TYPE UDT 31
VERSION : 0.0
  STRUCT
   A_FD_OR : BYTE ;	//Feedrate override
   A_DriveEnable : BOOL ;	//Drive test movement enable
   A_AckFixedStop : BOOL ;	//Acknowledge fixed stop reached
   A_SensorFixedStop : BOOL ;	//Sensor fixed stop
   A_ASpDisable : BOOL ;	//Axis/spindle disable
   A_Follow_upMode : BOOL ;	//Follow-up mode
   A_PosMeas1 : BOOL ;	//Position measuring system 1
   A_PosMeas2 : BOOL ;	//Position measuring system 2
   A_ORactive : BOOL ;	//Override active
   A_SWCam : BOOL ;	//SW cam activation
   A_ContrEnable : BOOL ;	//Controller enable
   A_DelDTGSpReset : BOOL ;	//Delete distance to go/Spindle-Reset
   A_Clamp : BOOL ;	//Clamping in progress
   A_RefVal1 : BOOL ;	//Reference point value 1
   A_RefVal2 : BOOL ;	//Reference point value 2
   A_RefVal3 : BOOL ;	//Reference point value 3
   A_RefVal4 : BOOL ;	//Reference point value 4
   A_ExtZO : BOOL ;	//Import external ZO
   A_EnabTravFixedStop : BOOL ;	//Enable travel to fixed stop
   A_FixedFD1 : BOOL ;	//Activate fixed feed 1
   A_FixedFD2 : BOOL ;	//Activate fixed feed 2
   A_FixedFD3 : BOOL ;	//Activate fixed feed 3
   A_FixedFD4 : BOOL ;	//Activate fixed feed 4
   A_VelocSpeedLimit : BOOL ;	//Velocity/spindle speed limitation
   A_PrgtestAxRel : BOOL ;	// Program test axis/spindle release
   A_HW1 : BOOL ;	//Activate handwheel 1
   A_HW2 : BOOL ;	//Activate handwheel 2
   A_HW3 : BOOL ;	//Activate handwheel 3
   A_FDSpStop : BOOL ;	//Feed stop/spindle stop
   A_Disable : BOOL ;	//Traversing key disable
   A_RapidTrOR : BOOL ;	//Rapid traverse override
   A_Minus : BOOL ;	//Traversing key minus
   A_Plus : BOOL ;	//Traversing key plus
   A_INC1 : BOOL ;	//INC1
   A_INC10 : BOOL ;	//INC10
   A_INC100 : BOOL ;	//INC100
   A_INC1000 : BOOL ;	//INC1000
   A_INC10000 : BOOL ;	//INC10000
   A_INCVar : BOOL ;	//INC variable
   A_OEMAxis : BYTE ;	//OEM axis signals
   A_InvHWDirOfRot : BOOL ;	// Inverting handwheel direction of rotation
   f7_1 : BOOL ;
   f7_2 : BOOL ;
   f7_3 : BOOL ;
   f7_4 : BOOL ;
   f7_5 : BOOL ;
   f7_6 : BOOL ;
   f7_7 : BOOL ;
   A_NCASpChanA : BOOL ;	//Assign NC axis/spindle channel A
   A_NCASpChanB : BOOL ;	//Assign NC axis/spindle channel B
   A_NCASpChanC : BOOL ;	//Assign NC axis/spindle channel C
   A_NCASpChanD : BOOL ;	//Assign NC axis/spindle channel D
   A_NCASpStrobe : BOOL ;	//Activation of assignment with pos. edge
   f8_5 : BOOL ;
   f8_6 : BOOL ;
   A_PLCASp : BOOL ;	//Request PLC axis/spindle
   A_Para_A : BOOL ;	//Parameter block servo A
   A_Para_B : BOOL ;	//Parameter block servo B
   A_Para_C : BOOL ;	//Parameter block servo C
   A_LockParSetDef : BOOL ;	//Lock parameter set definition from NC
   f9_4 : BOOL ;
   f9_5 : BOOL ;
   f9_6 : BOOL ;
   f9_7 : BOOL ;
   A_REPOSDelay : BOOL ;	//REPOS DELAY
   f10_1 : BOOL ;
   f10_2 : BOOL ;
   f10_3 : BOOL ;
   f10_4 : BOOL ;
   f10_5 : BOOL ;
   f10_6 : BOOL ;
   f10_7 : BOOL ;
   A_StartBrakeTest : BOOL ;	// Start brake test
   f11_1 : BOOL ;
   f11_2 : BOOL ;
   f11_3 : BOOL ;
   f11_4 : BOOL ;
   f11_5 : BOOL ;
   f11_6 : BOOL ;
   f11_7 : BOOL ;
   A_HWLimitMinus : BOOL ;	//Hardware limit switch minus
   A_HWLimitPlus : BOOL ;	//Hardware limit switch plus
   A_SWLimit2Minus : BOOL ;	//2nd software limit switch minus
   A_SWLimit2Plus : BOOL ;	//2nd software limit switch plus
   A_ModuloLimitEn : BOOL ;	// Modulo limit enabled
   f12_5 : BOOL ;
   f12_6 : BOOL ;
   A_DelayRef : BOOL ;	//Delay reference point approach
   A_JogFixPPos0 : BOOL ;	// JogFixPointPos 0
   A_JogFixPPos1 : BOOL ;	// JogFixPointPos 1
   A_JogFixPPos2 : BOOL ;	// JogFixPointPos 2
   A_JogToPos : BOOL ;	// Jog to position
   f13_4 : BOOL ;
   f13_5 : BOOL ;
   f13_6 : BOOL ;
   f13_7 : BOOL ;
   A_ProgtestSuppress : BOOL ;	// Program test to supress
   A_ProgtestActivate : BOOL ;	// Program test activate
   f14_2 : BOOL ;
   f14_3 : BOOL ;
   f14_4 : BOOL ;
   f14_5 : BOOL ;
   f14_6 : BOOL ;
   f14_7 : BOOL ;
   f15 : BYTE ;
   A_ActGearA : BOOL ;	//Actual gear stage A
   A_ActGearB : BOOL ;	//Actual gear stage B
   A_ActGearC : BOOL ;	//Actual gear stage C
   A_GearChangeOv : BOOL ;	//Gear has changed over
   A_Sp1Syn : BOOL ;	//Re-synchronize spindle 1
   A_Sp2Syn : BOOL ;	//Re-synchronize spindle 2
   A_NoMonitorGear : BOOL ;	//No monitoring when changing gear
   A_DeleteS : BOOL ;	//Delete S value
   A_FD_ORSp : BOOL ;	//Feedrate override for spindle valid
   f17_1 : BOOL ;
   f17_2 : BOOL ;
   f17_3 : BOOL ;
   A_Sp1SynP : BOOL ;	//Re-synchronize spindle 1 f. positioning
   A_Sp2SynP : BOOL ;	//Re-synchronize spindle 2 f. positioning
   A_M3M4Inv : BOOL ;	//Invert M3/M4
   f17_7 : BOOL ;
   f18_0 : BOOL ;
   f18_1 : BOOL ;
   f18_2 : BOOL ;
   f18_3 : BOOL ;
   A_OscilPLC : BOOL ;	//Oscillation via PLC
   A_OscilSpeed : BOOL ;	//enable Oscillation
   A_SetRotDirectRight : BOOL ;	//Setpoint osci. direct. right
   A_SetRotDirectLeft : BOOL ;	//Setpoint osci. direct. left
   A_SpOR : BYTE ;	//Spindle override
   f20_0 : BOOL ;
   A_RUEncQuStop : BOOL ;	//Run-up encoder quick stop
   f20_2 : BOOL ;
   A_SpeedSetpSmooth : BOOL ;	//Speed setpoint smoothing
   f20_4 : BOOL ;
   A_HoldBrakeToOpen : BOOL ;	// holding brake open
   f20_6 : BOOL ;
   f20_7 : BOOL ;
   A_ParA : BOOL ;	//Parameter set selection A
   A_ParB : BOOL ;	//Parameter set selection B
   A_ParC : BOOL ;	//Parameter set selection C
   A_MotA : BOOL ;	//Motor selection A
   A_MotB : BOOL ;	//Motor selection B
   A_MotOK : BOOL ;	//Motor selected
   A_IntegratDisable : BOOL ;	//n controller integrator disable
   A_PulseEnable : BOOL ;	//Pulse enable
   A_SG_SBH : BOOL ;	//Deselection SG/SBH
   A_SBH : BOOL ;	//Deselection of safe standstill
   f22_2 : BOOL ;
   A_SGselect0 : BOOL ;	//Selection SG bit 0
   A_SGselect1 : BOOL ;	//Selection SG bit 1
   f22_5 : BOOL ;
   f22_6 : BOOL ;
   f22_7 : BOOL ;
   A_Transmiss0 : BOOL ;	//Selection Transmission bit 0
   A_Transmiss1 : BOOL ;	//Selection Transmission bit 1
   A_Transmiss2 : BOOL ;	//Selection Transmission bit 2
   f23_3 : BOOL ;
   A_SE : BOOL ;	//Selection SE
   A_BrakeToClose : BOOL ;	//Sinamics: Brake to close
   f23_6 : BOOL ;
   A_TestStop : BOOL ;	//Activate test stop
   A_RotationMonit : BOOL ;	// Stepper motor: Rotation monitoring
   A_ControlAx : BOOL ;	// Control Axis
   f24_2 : BOOL ;
   f24_3 : BOOL ;
   A_TorqComp : BOOL ;	// Torque compensation
   A_ChangSetpOutAss0 : BOOL ;	// Bit value for CTRLOUT_changed - Change setpoint output assignment
   A_ChangSetpOutAss1 : BOOL ;	// Bit value for CTRLOUT_changed - Change setpoint output assignment
   A_MS : BOOL ;	//Master / Slave On
   A_DynBComp : BOOL ;	// dynamic backlash compensation activated
   f25_1 : BOOL ;
   f25_2 : BOOL ;
   f25_3 : BOOL ;
   f25_4 : BOOL ;
   f25_5 : BOOL ;
   f25_6 : BOOL ;
   f25_7 : BOOL ;
   f26_0 : BOOL ;
   f26_1 : BOOL ;
   f26_2 : BOOL ;
   A_CompContr : BOOL ;	//Compensation controller On
   A_FollowAxOv : BOOL ;	//Enable following axis override
   f26_5 : BOOL ;
   f26_6 : BOOL ;
   f26_7 : BOOL ;
   A_DEPMCS : BOOL ;	// Resume: DEPMCS
   A_DEPBCS : BOOL ;	// Resume: DEPBCS
   A_Corr : BOOL ;	// Resume: Corr
   A_HIAxMove : BOOL ;	// Resume: HIAxMove
   A_StopDEPMCS : BOOL ;	// Stop: DEPMCS
   A_StopDEPBCS : BOOL ;	// Stop: DEPBCS
   A_StopCorr : BOOL ;	// Stop: Corr
   A_StopHIAxMove : BOOL ;	// Stop: HIAxMove
   A_OscillAxExtRev : BOOL ;	// OscillAxExtReversal
   A_AxReset : BOOL ;	// AXRESET
   A_AxResume : BOOL ;	// AXRESUME
   A_SetRP : BOOL ;	//Set reversal point
   A_ChangeRP : BOOL ;	//Change reversal point
   A_StopRP : BOOL ;	//Stop at next reversal point
   A_Stop : BOOL ;	//Stop
   A_PLCAxis : BOOL ;	//PLC checks axis
   f29_0 : BOOL ;
   f29_1 : BOOL ;
   f29_2 : BOOL ;
   f29_3 : BOOL ;
   A_StartGantSynRun : BOOL ;	//Start gantry synchronization run
   A_NoAutoSync : BOOL ;	//No auto sync
   f29_6 : BOOL ;
   f29_7 : BOOL ;
   A_StopSpindle : BOOL ;	//Stop spindle
   A_StartCW : BOOL ;	//Start spindle Clockwise
   A_StartCCW : BOOL ;	//Start spindle Counterclockwise
   A_AutoGearStep : BOOL ;	//Autom. gear step change
   A_PosSpindle : BOOL ;	//Position spindle
   f30_5 : BOOL ;
   f30_6 : BOOL ;
   f30_7 : BOOL ;
   f31_0 : BOOL ;
   f31_1 : BOOL ;
   f31_2 : BOOL ;
   f31_3 : BOOL ;
   A_Resynchronize : BOOL ;	// Resynchronize
   A_DisSync : BOOL ;	// Disable synchronization
   A_Tracksync : BOOL ;	// Track synchronism
   A_DelSyncRunCorr : BOOL ;	// Deleting synchronous run correction
   f32_0 : BOOL ;
   f32_1 : BOOL ;
   A_extStopA : BOOL ;	//Deselection external Stop A
   A_extStopC : BOOL ;	//Deselection external Stop C
   A_extStopD : BOOL ;	//Deselection external Stop D
   A_extStopE : BOOL ;	//Deselection external Stop E
   f32_6 : BOOL ;
   f32_7 : BOOL ;
   f33_0 : BOOL ;
   f33_1 : BOOL ;
   f33_2 : BOOL ;
   f33_3 : BOOL ;
   A_SGcorr_0 : BOOL ;	//Selection SG-correction Bit 0
   A_SGcorr_1 : BOOL ;	//Selection SG-correction Bit 1
   A_SGcorr_2 : BOOL ;	//Selection SG-correction Bit 2
   A_SGcorr_3 : BOOL ;	//Selection SG-correction Bit 3
   A_SI_SetpLimBit0 : BOOL ;	// Set point limitation Bit0
   A_SI_SetpLimBit1 : BOOL ;	// Set point limitation Bit1
   f34_2 : BOOL ;
   f34_3 : BOOL ;
   f34_4 : BOOL ;
   f34_5 : BOOL ;
   f34_6 : BOOL ;
   f34_7 : BOOL ;
   f35 : BYTE ;
   f36 : ARRAY  [36 .. 55 ] OF BYTE ;
   A_FeedDriveCAxEng : BOOL ;	// Seperate feed drive as C axis engaged
   A_SpSpeedDisp : BOOL ;	// Spindle speed display
   A_SpInsideClamp : BOOL ;	// Spindle inside clamping
   f56_3 : BOOL ;
   f56_4 : BOOL ;
   f56_5 : BOOL ;
   f56_6 : BOOL ;
   f56_7 : BOOL ;
   f57 : BYTE ;
   f58 : WORD ;	// FC18: internal
   E_SpNA : BOOL ;	//Spindle/no axis
   E_NCU_Link : BOOL ;	//NCU_link active axis
   E_EncodFreq1 : BOOL ;	//Encoder limit frequency 1 exceeded
   E_EncodFreq2 : BOOL ;	//Encoder limit frequency 2 exceeded
   E_RefSyn1 : BOOL ;	//Referenced/synchronized 1
   E_RefSyn2 : BOOL ;	//Referenced/synchronized 2
   E_ExactCoarse : BOOL ;	//Position reached with exact stop coarse
   E_ExactFine : BOOL ;	//Position reached with exact stop fine
   E_TravRequ : BOOL ;	//Travel request
   E_AxialAlarm : BOOL ;	// Axial alarm
   E_AxisReady : BOOL ;	//Axis ready
   E_Follow_upMode : BOOL ;	//Follow-up mode active
   E_Stat : BOOL ;	//Axis/spindle stationary (n<nmin)
   E_PositContr : BOOL ;	//Position controller active
   E_SpeedContr : BOOL ;	//Speed controller active
   E_CurrentContr : BOOL ;	//Current controller active
   E_SWCam : BOOL ;	//Software cams active
   E_HWOverlay : BOOL ;	//Handwheel overlay active
   E_RevFD : BOOL ;	//Revolutional feedrate active
   E_MeasAct : BOOL ;	//Measuring active
   E_ActTravFStop : BOOL ;	//Activate travel to fixed stop
   E_FixedStop : BOOL ;	//Fixed stop reached
   E_ForceFixedStop : BOOL ;	// Force fixed stop limited
   E_AxContainerRot : BOOL ;	// Axis container rotation active
   E_AxReset : BOOL ;	// Axis reset done
   E_PLCCtrlAx : BOOL ;	// PLCcontrolled axis
   E_AxStop : BOOL ;	// Axis stop active
   E_AxSpDisable : BOOL ;	// Axis/spindle disable active
   E_StopDEPMCS : BOOL ;	// stop DEPMCS active
   E_StopDEPBCS : BOOL ;	// stop DEPBCS active
   E_StopCorr : BOOL ;	// stop Corr active
   E_StopHIAxMove : BOOL ;	// Stop HIAxMove active
   E_HW1 : BOOL ;	//Handwheel 1 active
   E_HW2 : BOOL ;	//Handwheel 2 active
   E_HW3 : BOOL ;	//Handwheel 3 active
   f64_3 : BOOL ;
   E_TReqMinus : BOOL ;	// Travel request minus
   E_TReqPlus : BOOL ;	// Travel request plus
   E_TCMinus : BOOL ;	//Traverse command minus
   E_TCPlus : BOOL ;	//Traverse command plus
   E_INC1 : BOOL ;	//INC1
   E_INC10 : BOOL ;	//INC10
   E_INC100 : BOOL ;	//INC100
   E_INC1000 : BOOL ;	//INC1000
   E_INC10000 : BOOL ;	//INC10000
   E_INCVar : BOOL ;	//INC variable
   f65_6 : BOOL ;
   f65_7 : BOOL ;
   E_OEMAxis : BYTE ;	//OEM axis signals
   E_InvHWDirOfRot : BOOL ;	// Handwheel direction of rotation invert actively
   f67_1 : BOOL ;
   f67_2 : BOOL ;
   f67_3 : BOOL ;
   f67_4 : BOOL ;
   f67_5 : BOOL ;
   f67_6 : BOOL ;
   f67_7 : BOOL ;
   E_NCASpChanA : BOOL ;	//NC axis/spindle in channel A
   E_NCASpChanB : BOOL ;	//NC axis/spindle in channel B
   E_NCASpChanC : BOOL ;	//NC axis/spindle in channel C
   E_NCASpChanD : BOOL ;	//NC axis/spindle in channel D
   E_PLCType : BOOL ;	//New type requested by PLC
   E_ChPoss : BOOL ;	//Change axis possible
   E_NeutrASp : BOOL ;	//Neutral axis/spindle
   E_PLCASp : BOOL ;	//PLC axis/spindle
   E_ParS_A : BOOL ;	//Parameter block servo A
   E_ParS_B : BOOL ;	//Parameter block servo B
   E_ParS_C : BOOL ;	//Parameter block servo C
   E_NCUNumLink_3 : BOOL ;
   E_NCUNumLink_4 : BOOL ;
   E_NCUNumLink_5 : BOOL ;
   E_NCUNumLink_6 : BOOL ;
   E_NCUNumLink_7 : BOOL ;
   E_ReposSh : BOOL ;	// Repos shift
   E_ReposShValid : BOOL ;	// Repos shift valid
   E_ReposDelayQuit : BOOL ;	// Repos delay quit
   f70_3 : BOOL ;
   E_SI_Nck : BOOL ;	// NCK-Safety Integrated active
   E_SI_Drv_SICSCC : BOOL ;	// DRV-Safety Integrated with SIC/SCC active
   f70_6 : BOOL ;
   f70_7 : BOOL ;
   E_BrakeTest : BOOL ;	// Brake test active
   f71_1 : BOOL ;
   f71_2 : BOOL ;
   f71_3 : BOOL ;
   E_POS_RESTORED1 : BOOL ;	// POS_RESTORED 1
   E_POS_RESTORED2 : BOOL ;	// POS_RESTORED 2
   f71_6 : BOOL ;
   E_PLCAxDedic : BOOL ;	// PLC Axis dedicated
   E_MMC_REPOSDelay : BOOL ;	//MMC REPOS DELAY
   f72_1 : BOOL ;
   f72_2 : BOOL ;
   f72_3 : BOOL ;
   f72_4 : BOOL ;
   f72_5 : BOOL ;
   f72_6 : BOOL ;
   f72_7 : BOOL ;
   f73 : BYTE ;
   f74_0 : BOOL ;
   f74_1 : BOOL ;
   f74_2 : BOOL ;
   f74_3 : BOOL ;
   E_ModLimEnAct : BOOL ;	// Modulo limit enabled active
   f74_5 : BOOL ;
   f74_6 : BOOL ;
   f74_7 : BOOL ;
   E_JogFixPPos0Act : BOOL ;	// JogFixPointPos 0 active
   E_JogFixPPos1Act : BOOL ;	// JogFixPointPos 1 active
   E_JogFixPPos2Act : BOOL ;	// JogFixPointPos 2 active
   E_JogFixPPos0 : BOOL ;	// JogFixPointPos 0 reached
   E_JogFixPPos1 : BOOL ;	// JogFixPointPos 1 reached
   E_JogFixPPos2 : BOOL ;	// JogFixPointPos 2 reached
   E_JogToPos : BOOL ;	// Jog to position active
   E_JogPos : BOOL ;	// Jog position reached
   E_ScratchPulse : BOOL ;	//Scratch pulse
   f76_1 : BOOL ;
   f76_2 : BOOL ;
   f76_3 : BOOL ;
   E_PathAxis : BOOL ;	// Path axis
   E_PosAxis : BOOL ;	//Positioning axis
   E_IndexAxisPos : BOOL ;	//Indexing axis in position
   E_CurvePos : BOOL ;	//Curve axis in position
   E_CollCheckRedSpeed : BOOL ;	//reduced speed of Collisions Check
   f77_1 : BOOL ;
   f77_2 : BOOL ;
   f77_3 : BOOL ;
   f77_4 : BOOL ;
   f77_5 : BOOL ;
   f77_6 : BOOL ;
   f77_7 : BOOL ;
   E_FPosAxis : REAL ;	//F function (REAL format) for positioning axes
   E_SetpGearA : BOOL ;	//Setpoint gear stage A
   E_SetpGearB : BOOL ;	//Setpoint gear stage B
   E_SetpGearC : BOOL ;	//Setpoint gear stage C
   E_GearChange : BOOL ;	//Gear changeover
   f82_4 : BOOL ;
   f82_5 : BOOL ;
   f82_6 : BOOL ;
   f82_7 : BOOL ;
   E_SpeedLimit : BOOL ;	//Speed limit exceeded
   E_SetSpeedLimit : BOOL ;	//Setpoint speed limited
   E_SetSpeedIncreased : BOOL ;	//Setpoint speed increased
   E_GeoMonit : BOOL ;	//Geometry monitoring
   E_SupportAreaViol : BOOL ;	//Support area limits violated
   E_SetRange : BOOL ;	//Spindle in setpoint range
   E_SpeedMonit : BOOL ;	//Speed monitoring
   E_ActRotRight : BOOL ;	//Actual rotation direction right
   E_ConstCuttSpeed : BOOL ;	//Const. cutting speed active
   E_SUG : BOOL ;	//SUG active (grinding wheel surface speed)
   E_CLG : BOOL ;	//CLG active
   E_Tapping : BOOL ;	//Tapping without compensating chuck
   E_SyncMode : BOOL ;	//Synchronous mode spindle active
   E_PosMode : BOOL ;	//Positioning mode spindle active
   E_OscillMode : BOOL ;	//Oscillation mode spindle active
   E_ContrMode : BOOL ;	//Control mode spindle active
   E_ToolDynLimit : BOOL ;	// Tool with limit of dynamics
   f85_1 : BOOL ;
   f85_2 : BOOL ;
   f85_3 : BOOL ;
   f85_4 : BOOL ;
   E_SpInPosition : BOOL ;	// Spindle in position
   f85_6 : BOOL ;
   f85_7 : BOOL ;
   E_MFunct : INT ;	//M function (INT) for spindle
   E_SFunct : REAL ;	//S function (REAL) for spindle
   f92_0 : BOOL ;
   E_RUEncDisabl : BOOL ;	//Run-up encoder disable active
   f92_2 : BOOL ;
   E_SpeedSetpSmooth : BOOL ;	//Speed setpoint smoothing active
   E_RLIact : BOOL ;	// RLI active
   E_HoldBrakeOpened : BOOL ;	// Holding brake opened
   f92_6 : BOOL ;
   E_DriveRunEn : BOOL ;	// Drive run enabled
   E_ParA : BOOL ;	//Active parameter set A
   E_ParB : BOOL ;	//Active parameter set B
   E_ParC : BOOL ;	//Active parameter set C
   E_MotA : BOOL ;	//Active motor A
   E_MotB : BOOL ;	//Active motor B
   E_MotOK : BOOL ;	//Drive ready
   E_IntegratDisable : BOOL ;	//n controller integrator disabled
   E_PulseEnable : BOOL ;	//Pulses enabled
   E_MTempWarn : BOOL ;	//Temperature prewarning motor
   E_HTempWarn : BOOL ;	//Temperature prewarning heat sink
   E_RUComplete : BOOL ;	//Ramp-up complete
   E_MdMdx : BOOL ;	//Md<Mdx
   E_NactNmin : BOOL ;	//nact<nmin
   E_NactNx : BOOL ;	//nact<nx
   E_NactNset : BOOL ;	//nact=nset
   E_Message : BOOL ;	//Variable message function
   E_UDClessAlThreshold : BOOL ;	//UDC-link < alarm threshold
   f95_1 : BOOL ;
   f95_2 : BOOL ;
   f95_3 : BOOL ;
   f95_4 : BOOL ;
   f95_5 : BOOL ;
   f95_6 : BOOL ;
   E_I2TLimit : BOOL ;	// Power Section I2T limit
   E_SpindleMonit : BOOL ;	//Error spindle monitoring
   E_AxisCtrl : BOOL ;	// Axis control active
   E_MSFine : BOOL ;	// Master/Slave fine
   E_MSCoarse : BOOL ;	// Master/Slave coarse
   E_MSCompContr : BOOL ;	// Master/Slave Compensation controller activ
   E_BitValCtrlOutChang0 : BOOL ;	// Bit value for CTRLOUT_changed 0:  Change setpoint output assignment
   E_BitValCtrlOutChang1 : BOOL ;	// Bit value for CTRLOUT_changed 1:  Change setpoint output assignment
   E_MS : BOOL ;	//Master/ slave active
   f97 : BYTE ;
   E_SyncronFine : BOOL ;	//Synchronism fine
   E_SyncronCoarse : BOOL ;	//Synchronism coarse
   E_ActValCoupling : BOOL ;	//Actual value coupling
   f98_3 : BOOL ;
   E_OverlayMotion : BOOL ;	//Overlaid motion
   E_SWL : BOOL ;	//Speed warning limit reached
   E_AWL : BOOL ;	//Acceleration warning limit reached
   E_EmRetr : BOOL ;	//Emergency retraction active
   E_MasterSp : BOOL ;	//Master spindle
   E_SlaveSp : BOOL ;	//Slave spindle
   E_SyncRunCorrDOut : BOOL ;	// Synchronous run correction driven out
   E_AxisAccel : BOOL ;	//Axis accelerated
   E_Sync : BOOL ;	//Synchronization active
   E_MSR : BOOL ;	//Max speed reached
   E_MAR : BOOL ;	//Max acceleration reached
   f99_7 : BOOL ;
   f100_0 : BOOL ;
   f100_1 : BOOL ;
   E_OscillAxExtRev : BOOL ;	// OscillAxExt Reversal active
   E_StopOscill : BOOL ;	//Oscillation cannot start
   E_ErrorOscill : BOOL ;	//Error during oscillation
   E_SparkOut : BOOL ;	//Spark-out active
   E_OscillMotion : BOOL ;	//Oscillation motion active
   E_Oscill : BOOL ;	//Oscillation active
   f101_0 : BOOL ;
   f101_1 : BOOL ;
   E_GantCOLimit : BOOL ;	//Gantry cut-off limit exceeded
   E_GantWarn : BOOL ;	//Gantry warning limit exceeded
   E_SynRunStart : BOOL ;	//Synchronization run ready to start
   E_GantGroupSyn : BOOL ;	//Gantry grouping is synchronous
   E_GantLeadAxis : BOOL ;	//Gantry leading axis
   E_GantAxis : BOOL ;	//Gantry axis
   E_DynBComp : BOOL ;	// dynamic backlash compensation activ
   f102_1 : BOOL ;
   f102_2 : BOOL ;
   f102_3 : BOOL ;
   f102_4 : BOOL ;
   f102_5 : BOOL ;
   f102_6 : BOOL ;
   f102_7 : BOOL ;
   E_SyncRunCorrIncl : BOOL ;	// Synchronous run correction is included
   f103_1 : BOOL ;
   f103_2 : BOOL ;
   f103_3 : BOOL ;
   E_Syncron2Fine : BOOL ;	//Synchronism fine
   E_Syncron2Coarse : BOOL ;	//Synchronism coarse
   f103_6 : BOOL ;
   f103_7 : BOOL ;
   E_AIAxis : ARRAY  [1 .. 31 ] OF BOOL ;	//Active infeed axis[1..31]
   E_SG_SBH : BOOL ;	//Active SG/SBH
   E_ErrLifeS_CRC : BOOL ;	// Error lifesign or CRC-error
   E_ImpdelNCK : BOOL ;	//Delete pulses NCK
   r108_3 : BOOL ;
   r108_4 : BOOL ;
   r108_5 : BOOL ;
   r108_6 : BOOL ;
   E_SRef : BOOL ;	//Axis safely referenced
   E_SN1Plus : BOOL ;	//Actual position > cam position SN1+
   E_SN1Minus : BOOL ;	//Actual position > cam position SN1-
   E_SN2Plus : BOOL ;	//Actual position > cam position SN2+
   E_SN2Minus : BOOL ;	//Actual position > cam position SN2-
   E_SN3Plus : BOOL ;	//Actual position > cam position SN3+
   E_SN3Minus : BOOL ;	//Actual position > cam position SN3-
   E_SN4Plus : BOOL ;	//Actual position > cam position SN4+
   E_SN4Minus : BOOL ;	//Actual position > cam position SN4-
   f110_0 : BOOL ;
   E_SBH : BOOL ;	//Active SBH
   f110_2 : BOOL ;
   E_SG_0 : BOOL ;	//Active SG 0
   E_SG_1 : BOOL ;	//Active SG 1
   E_n_nx : BOOL ;	//n < nx
   f110_6 : BOOL ;
   f110_7 : BOOL ;
   f111_0 : BOOL ;
   f111_1 : BOOL ;
   f111_2 : BOOL ;
   f111_3 : BOOL ;
   E_StopAB : BOOL ;	//Stop A/B active
   E_StopC : BOOL ;	//Stop C active
   E_StopD : BOOL ;	//Stop D active
   E_StopE : BOOL ;	//Stop E active
   E_CamRangeTr1 : BYTE ;	//Cam Range for Cam Track 1
   E_CamRangeTr2 : BYTE ;	//Cam Range for Cam Track 2
   E_CamRangeTr3 : BYTE ;	//Cam Range for Cam Track 3
   E_CamRangeTr4 : BYTE ;	//Cam Range for Cam Track 4
   f116 : BYTE ;
   E_CamTrack1 : BOOL ;	//Cam Track 1
   E_CamTrack2 : BOOL ;	//Cam Track 2
   E_CamTrack3 : BOOL ;	//Cam Track 3
   E_CamTrack4 : BOOL ;	//Cam Track 4
   f117_4 : BOOL ;
   f117_5 : BOOL ;
   f117_6 : BOOL ;
   f117_7 : BOOL ;
   E_CamRangeBitTr1 : ARRAY  [0 .. 14 ] OF //Cam Range Bits for Cam Track 1
   BOOL ;
   E_CamRangeBitTr2 : ARRAY  [0 .. 14 ] OF //Cam Range Bits for Cam Track 2
   BOOL ;
   E_CamRangeBitTr3 : ARRAY  [0 .. 14 ] OF //Cam Range Bits for Cam Track 3
   BOOL ;
   E_CamRangeBitTr4 : ARRAY  [0 .. 14 ] OF //Cam Range Bits for Cam Track 4
   BOOL ;
   f126 : WORD ;	// internal
   E_MMC_ProgtestSuppress : BOOL ;	// HMI->PLC: Program test to supress
   E_MMC_ProgtestActivate : BOOL ;	// HMI->PLC: Program test activate
   f128_2 : BOOL ;
   f128_3 : BOOL ;
   f128_4 : BOOL ;
   f128_5 : BOOL ;
   f128_6 : BOOL ;
   f128_7 : BOOL ;
   f129 : BYTE ;
   f130 : WORD ;
   E_SensorAv : BOOL ;	// Sensors available
   E_S1aMeasARod : BOOL ;	// Sensor S1: analogous measurement position of actuating rod
   f132_2 : BOOL ;
   f132_3 : BOOL ;
   E_S4dPistonStopP : BOOL ;	// Sensor S4: digital value piston stop position
   E_S5dAngleShaft : BOOL ;	// Sensor S5: digital value angle situation shaft
   E_S6Temp : BOOL ;	// Sensor S6:temperature
   f132_7 : BOOL ;
   f133 : BYTE ;
   E_ClampingState : INT ;	// state of the clamping system
   E_AnalogSensor : INT ;	// analog sensor on the motor
   f138_0 : BOOL ;
   f138_1 : BOOL ;
   f138_2 : BOOL ;
   f138_3 : BOOL ;
   E_S4PistonStopP : BOOL ;	// Sensor S4: piston stop position
   E_S5AngleShaft : BOOL ;	// Sensor S5: angle situation shaft
   f138_6 : BOOL ;
   f138_7 : BOOL ;
   f139 : BYTE ;
  END_STRUCT ;	
END_TYPE

TYPE UDT 71
VERSION : 0.0
  STRUCT
   IFNo : ARRAY  [1 .. 16 ] OF BOOL ;	//Interface [no.] active
   Quit : ARRAY  [1 .. 16 ] OF BOOL ;	//perform Quit-End
   IF : ARRAY  [1 .. 16 ] OF STRUCT
    Loading : BOOL ;
    Unloading : BOOL ;
    Reloading : BOOL ;
    Positioning : BOOL ;
    PosbyProgram : BOOL ;	//Initiation by CNC Program
    PositioningMT : BOOL ;	//Positioning Multitool
    f0_6 : BOOL ;
    f0_7 : BOOL ;
    PerfStatusError : BOOL ;
    n1_1 : BOOL ;
    n1_2 : BOOL ;
    n1_3 : BOOL ;
    n1_4 : BOOL ;
    n1_5 : BOOL ;
    n1_6 : BOOL ;
    DataInDB1071 : BOOL ;
    Channel : BYTE ;	//Assigned channel
    TMno : BYTE ;	//Tool management no.
    Free1 : DINT ;	//Unassigned parameter 1
    Free2 : DINT ;	//Unassigned parameter 2
    Free3 : DINT ;	//Unassigned parameter 3
    IdentLoad : INT ;	//Identification for loading/unloading station
    NoLoad : INT ;	//No. of loading station
    SMag : INT ;	//Magazine no. (source) for unloading/reloading/pos.
    SLoc : INT ;	//Location no. (source) for unloading/reloading/pos.
    TMag : INT ;	//Magazine no. (target) for loading/reloading
    TLoc : INT ;	//Location no. (target) for loading/reloading
    WithoutMagMoving : BOOL ;	//HMI Data: Without Magazine Moving
    Res2 : BYTE ;
   END_STRUCT ;
  END_STRUCT ;	
END_TYPE

TYPE UDT 72
VERSION : 0.0
  STRUCT
   IFNo : ARRAY  [1 .. 16 ] OF BOOL ;	//Interface [no.] active
   Quit : ARRAY  [1 .. 16 ] OF BOOL ;	//perform Quit-End
   IF : ARRAY  [1 .. 16 ] OF STRUCT
    Comp : BOOL ;	//Compulsory change
    Perform : BOOL ;	//Perform change
    Prepare : BOOL ;	//Prepare change
    T0 : BOOL ;	//T0 programmed
    OldTinDBW42 : BOOL ;	//ZWS No. of Old Tool in DBW (n+42)
    ManTIn : BOOL ;	//Put in Tool in Spindle manual
    ManTOut : BOOL ;	//Get out Tool from Spindle manual
    SpiTRSpi : BOOL ;	//Spindle Tool remains in spindle
    PerfStatusError : BOOL ;
    n1_1 : BOOL ;
    n1_2 : BOOL ;
    n1_3 : BOOL ;
    n1_4 : BOOL ;
    n1_5 : BOOL ;
    n1_6 : BOOL ;
    DataInDB1072 : BOOL ;
    Channel : BYTE ;	//Assigned channel
    TMno : BYTE ;	//Tool management no.
    Free1 : DINT ;	//Unassigned parameter 1
    Free2 : DINT ;	//Unassigned parameter 2
    Free3 : DINT ;	//Unassigned parameter 3
    IdentBuff : INT ;	//Buffer identification (fixed value 9998)
    NoBuff : INT ;	//Relative location (target) in the buffer
    SMag : INT ;	//Magazine no. (source) for new tool
    SLoc : INT ;	//Location no. (source) for new tool
    TMag : INT ;	//Magazine no. (target) for old tool
    TLoc : INT ;	//Location no. (target) for old tool
    LocType : INT ;	//Tool new: location type
    SLeft : INT ;	//Tool new: size left
    SRight : INT ;	//Tool new: size right
    STop : INT ;	//Tool new: size top
    SBottom : INT ;	//Tool new: size bottom
    ToolInBuff : BOOL ;	//ID for tools in buffer
    IgnoreDisab : BOOL ;	//Ignore disabled
    TBUnloaded : BOOL ;	//To be unloaded
    TBLoaded : BOOL ;	//To be loaded
    MasterTool : BOOL ;	//Master tool
    n38_5 : BOOL ;	//reserved
    Exchange_1to1 : BOOL ;	//1:1 exchange
    HandTool : BOOL ;	//Hand tool
    ActTool : BOOL ;	//Active tool
    ToolEnabl : BOOL ;	//Tool enabled
    ToolDisab : BOOL ;	//Tool disabled
    Measured : BOOL ;	//Tool measured
    Prewarn : BOOL ;	//Prewarning limit reached
    ToolChange : BOOL ;	//Tool being changed
    FixedLoc : BOOL ;	//Tool fixed location coded
    ToolUsed : BOOL ;	//Tool was in use
    T_no : INT ;	//Tool new: T no.
    OldTZWSNo : INT ;	//ZWS No. of Old Tool
    MyMag : INT ;
    MyPlace : INT ;
   END_STRUCT ;
  END_STRUCT ;	
END_TYPE

TYPE UDT 73
VERSION : 0.0
  STRUCT
   IfNo : ARRAY  [1 .. 16 ] OF BOOL ;	//Interface [no.] active
   Quit : ARRAY  [1 .. 16 ] OF BOOL ;	//perform Quit-End
   IF : ARRAY  [1 .. 16 ] OF STRUCT
    Comp : BOOL ;	//Compulsory change
    Perform : BOOL ;	//Perform change
    f0_2 : BOOL ;
    T0 : BOOL ;	//T0 programmed
    f0_4 : BOOL ;
    f0_5 : BOOL ;
    ManTOut : BOOL ;	//Get out Tool from Holder manual
    f0_7 : BOOL ;
    PerfStatusError : BOOL ;
    n1_1 : BOOL ;
    n1_2 : BOOL ;
    n1_3 : BOOL ;
    n1_4 : BOOL ;
    n1_5 : BOOL ;
    n1_6 : BOOL ;
    DataInDB1073 : BOOL ;
    Channel : BYTE ;	//Assigned channel
    TMno : BYTE ;	//Tool management no.
    Free1 : DINT ;	//Unassigned parameter 1
    Free2 : DINT ;	//Unassigned parameter 2
    Free3 : DINT ;	//Unassigned parameter 3
    KennZWS : INT ;	//Reserved (buffer identification)
    NoBuff : INT ;	//Rel. location in buffer (res.)
    SMag : INT ;	//Magazine no. of turret
    SLoc : INT ;	//Location no. for new tool
    TMag : INT ;	//Magazine no. of turret (res.)
    TLoc : INT ;	//Location no. for old tool
    LocType : INT ;	//Tool new: location type
    SLeft : INT ;	//Tool new: size left
    SRight : INT ;	//Tool new: size right
    STop : INT ;	//Tool new: size top
    SBottom : INT ;	//Tool new: size bottom
    ToolInBuff : BOOL ;	//ID for tools in buffer
    IgnoreDisab : BOOL ;	//Ignore disabled
    TBUnloaded : BOOL ;	//To be unloaded
    TBLoaded : BOOL ;	//To be loaded
    MasterTool : BOOL ;	//Master tool
    n38_5 : BOOL ;	//reserved
    Exchange_1to1 : BOOL ;	//1:1 exchange
    HandTool : BOOL ;	//Hand tool
    ActTool : BOOL ;	//Active tool
    ToolEnabl : BOOL ;	//Tool enabled
    ToolDisab : BOOL ;	//Tool disabled
    Measured : BOOL ;	//Tool measured
    Prewarn : BOOL ;	//Prewarning limit reached
    ToolChange : BOOL ;	//Tool being changed
    FixedLoc : BOOL ;	//Tool fixed location coded
    ToolUsed : BOOL ;	//Tool was in use
    T_no : INT ;	//Tool new: T no.
    MyPlace : INT ;
   END_STRUCT ;
  END_STRUCT ;	
END_TYPE

TYPE UDT 77
VERSION : 0.0
  STRUCT
   MCP1In : ARRAY  [0 .. 7 ] OF BYTE ;
   MCP1Out : ARRAY  [0 .. 7 ] OF BYTE ;
   MCP1StatSend : DWORD ;
   MCP1StatRec : DWORD ;
   MCP2In : ARRAY  [0 .. 7 ] OF BYTE ;
   MCP2Out : ARRAY  [0 .. 7 ] OF BYTE ;
   MCP2StatSend : DWORD ;
   MCP2StatRec : DWORD ;
   BHGIn : ARRAY  [0 .. 5 ] OF BYTE ;
   Filler : ARRAY  [0 .. 5 ] OF BYTE ;
   BHGOut : ARRAY  [0 .. 19 ] OF BYTE ;
   BHGStatSend : DWORD ;
   BHGStatRec : DWORD ;
  END_STRUCT ;	
END_TYPE

TYPE UDT 1002
VERSION : 0.0
  STRUCT 	//Offset 0
   Chan : ARRAY  [1 .. 10 ] OF STRUCT 	//From Channel 1 to Channel 10
    FDD : ARRAY  [0 .. 15 ] OF //Feed disable
    BOOL ;
    RID : ARRAY  [0 .. 15 ] OF //Read-in disable
    BOOL ;
    NCSD : ARRAY  [0 .. 15 ] OF //NC start disable
    BOOL ;
    FdStop_1 : ARRAY  [0 .. 15 ] OF //Feed stop GEOaxis 1
    BOOL ;
    FdStop_2 : ARRAY  [0 .. 15 ] OF //Feed stop GEOaxis 2
    BOOL ;
    FdStop_3 : ARRAY  [0 .. 15 ] OF //Feed stop GEOaxis 3
    BOOL ;
   END_STRUCT ;	//without Alarmno for Chan (120 Byte)
//Offset 120
   Axis : ARRAY  [1 .. 31 ] OF STRUCT 	//From Axis 1 to Axis 31
    FdStop : ARRAY  [0 .. 15 ] OF //Feed stop axis/spindle 1
    BOOL ;
   END_STRUCT ;	//without Alarmno for Axis (62 Byte)
//Offset 182
   ZInfo0 : ARRAY  [0 .. 63 ] OF WORD ;	//Additional Value for UserAlarms 700000 to 700063
//Offset 310
   ChanA : ARRAY  [1 .. 10 ] OF STRUCT 	//From Channel 1 to Channel 10
    FDD_5C00xx : ARRAY  [0 .. 15 ] OF //Feed disable A.no.51000-510015
    BOOL ;
    FDD_RID_5C01xx : ARRAY  [0 .. 31 ] OF //Feed and read-in disable A.no.510100-510131
    BOOL ;
    RID_5C02xx : ARRAY  [0 .. 31 ] OF //Read-in disable A.no.510200-510231
    BOOL ;
    NCSD_5C03xx : ARRAY  [0 .. 15 ] OF //NC start disable A.no.510300-510315
    BOOL ;
    FdStop_1_5C11xx : ARRAY  [0 .. 15 ] OF //Feed stop GEOaxis 1 A.no.511100-511115
    BOOL ;
    FdStop_2_5C12xx : ARRAY  [0 .. 15 ] OF //Feed stop GEOaxis 2 A.no.511200-511215
    BOOL ;
    FdStop_3_5C13xx : ARRAY  [0 .. 15 ] OF //Feed stop GEOaxis 3 A.no.511300-511315
    BOOL ;
   END_STRUCT ;	//Alarmno for Chan are 5Cxxxx; C is the ChannelNo, except Channel 10. Channel 10
   AxisA : ARRAY  [1 .. 32 ] OF STRUCT 	//From Axis 1 to Axis 31
    AAFdStop60AAxx : ARRAY  [0 .. 15 ] OF //Feed stop axis/spindle
    BOOL ;
   END_STRUCT ;	//Alarmno for Axis are 60AAxx; A is the Axisno.
//Offset 554
   UserA : ARRAY  [0 .. 31 ] OF STRUCT
    A70UUxx : ARRAY  [0 .. 63 ] OF //Alarm 700000-700063 (user area 0)
    BOOL ;
   END_STRUCT ;	//Alarmno for UserAlarms are 7yUUxx; U is the Userarea, y = Db1004.UserDek2No[U]
  END_STRUCT ;	
END_TYPE

TYPE UDT 1071
VERSION : 0.0
  STRUCT
   MTIF : ARRAY  [1 .. 16 ] OF STRUCT
    MtType : INT ;
    MtPlaces : INT ;
    MtDistance : REAL ;
    MtNum : INT ;	// MT-No. to be positioned to
    MtPlaceNum : INT ;	// MT-PlaceNo. ~
    ToolHolder : INT ;	// TH-No as reference for MT-positioning
    IF : ARRAY  [1 .. 3 ] OF STRUCT
     reserved : INT ;	// reserved
    END_STRUCT ;
   END_STRUCT ;
  END_STRUCT ;	
END_TYPE

TYPE UDT 1072
VERSION : 0.0
  STRUCT
   MTIF : ARRAY  [1 .. 16 ] OF STRUCT
    MtType : INT ;
    MtPlaces : INT ;
    MtDistance : REAL ;
    MtNumNew : INT ;	// MT-No. new Tool
    MtPlaceNumNew : INT ;	// MtoolPlaceNum  ~
    MtNumOld : INT ;	// MT-No. old Tool
    MtPlaceNumOld : INT ;	// MtoolPlaceNum  ~
    LocType : INT ;	//Tool new: location type
    SLeft : INT ;	//Tool new: size left
    SRight : INT ;	//Tool new: size right
    STop : INT ;	//Tool new: size top
    SBottom : INT ;	//Tool new: size bottom
    ToolInBuff : BOOL ;	//ID for tools in buffer
    IgnoreDisab : BOOL ;	//Ignore disabled
    TBUnloaded : BOOL ;	//To be unloaded
    TBLoaded : BOOL ;	//To be loaded
    MasterTool : BOOL ;	//Master tool
    n26_5 : BOOL ;	//reserved
    n26_6 : BOOL ;	//reserved
    HandTool : BOOL ;	//Hand tool
    ActTool : BOOL ;	//Active tool
    ToolEnabl : BOOL ;	//Tool enabled
    ToolDisab : BOOL ;	//Tool disabled
    Measured : BOOL ;	//Tool measured
    Prewarn : BOOL ;	//Prewarning limit reached
    ToolChange : BOOL ;	//Tool being changed
    FixedLoc : BOOL ;	//Tool fixed location coded
    ToolUsed : BOOL ;	//Tool was in use
    T_no : INT ;	//Tool new: T no.
    ToolHolder : INT ;	// TH-No as tool compensation reference
    MtMyMag : INT ;	// MtoolNumber the tool is loaded onto
    MtMyPlace : INT ;	// MtoolPlaceNum ~
    IF : ARRAY  [1 .. 7 ] OF STRUCT
     reserved : INT ;	// reserved
    END_STRUCT ;
   END_STRUCT ;
  END_STRUCT ;	
END_TYPE

TYPE UDT 1073
VERSION : 0.0
  STRUCT
   MTIF : ARRAY  [1 .. 16 ] OF STRUCT
    MtType : INT ;
    MtPlaces : INT ;
    MtDistance : REAL ;
    MtNumNew : INT ;	// MT-No. new Tool
    MtPlaceNumNew : INT ;	// MtoolPlaceNum  ~
    MtNumOld : INT ;	// MT-No. old Tool
    MtPlaceNumOld : INT ;	// MtoolPlaceNum  ~
    LocType : INT ;	//Tool new: location type
    SLeft : INT ;	//Tool new: size left
    SRight : INT ;	//Tool new: size right
    STop : INT ;	//Tool new: size top
    SBottom : INT ;	//Tool new: size bottom
    ToolInBuff : BOOL ;	//ID for tools in buffer
    IgnoreDisab : BOOL ;	//Ignore disabled
    TBUnloaded : BOOL ;	//To be unloaded
    TBLoaded : BOOL ;	//To be loaded
    MasterTool : BOOL ;	//Master tool
    n26_5 : BOOL ;	//reserved
    n26_6 : BOOL ;	//reserved
    HandTool : BOOL ;	//Hand tool
    ActTool : BOOL ;	//Active tool
    ToolEnabl : BOOL ;	//Tool enabled
    ToolDisab : BOOL ;	//Tool disabled
    Measured : BOOL ;	//Tool measured
    Prewarn : BOOL ;	//Prewarning limit reached
    ToolChange : BOOL ;	//Tool being changed
    FixedLoc : BOOL ;	//Tool fixed location coded
    ToolUsed : BOOL ;	//Tool was in use
    T_no : INT ;	//Tool new: T no.
    ToolHolder : INT ;	// TH-No as tool compensation reference
    MtMyMag : INT ;	// MtoolNumber the tool is loaded onto
    MtMyPlace : INT ;	// MtoolPlaceNum ~
    IF : ARRAY  [1 .. 7 ] OF STRUCT
     reserved : INT ;	// reserved
    END_STRUCT ;
   END_STRUCT ;
  END_STRUCT ;	
END_TYPE

// FB 1: know-how protected block, not included

// FB 2: know-how protected block, not included

// FB 3: know-how protected block, not included

// FB 4: know-how protected block, not included

// FB 5: know-how protected block, not included

// FB 7: know-how protected block, not included

// FB 9: know-how protected block, not included

// FB 10: know-how protected block, not included

// FB 11: know-how protected block, not included

// FB 29: know-how protected block, not included

// FC 2: know-how protected block, not included

// FC 3: know-how protected block, not included

// FC 5: know-how protected block, not included

// FC 6: know-how protected block, not included

// FC 7: know-how protected block, not included

// FC 8: know-how protected block, not included

// FC 9: know-how protected block, not included

// FC 10: know-how protected block, not included

FUNCTION FC 12 : VOID
AUTHOR : NUMERIK
FAMILY : _800D
NAME : Basics
VERSION : 4.5
VAR_INPUT
  Chan : BYTE ;	//Index of Chan
END_VAR
BEGIN
// (block stored without names or comments; labels and parameter names are numbered)
END_FUNCTION

// FC 13: know-how protected block, not included

// FC 17: know-how protected block, not included

// FC 18: know-how protected block, not included

// FC 19: know-how protected block, not included

// FC 21: know-how protected block, not included

// FC 22: know-how protected block, not included

// FC 24: know-how protected block, not included

// FC 25: know-how protected block, not included

// FC 26: know-how protected block, not included

FUNCTION "Functions block call" : VOID	// FC 29
//KNOW_HOW_PROTECT
//
VERSION : 0.1
BEGIN
NETWORK
TITLE =
      CALL  "Enable_Control";
      CALL  "All motors_ control";
      CALL  "NC AND PLC CHANGE DATA";
      CALL  "HandWheelUnit_Control";
      CALL  "System_Date";
      CALL  "X_BACK_Control";
      CALL  "Grinding_Speed_2";
      BE;
END_FUNCTION

FUNCTION "Enable_Control" : VOID	// FC 30
//KNOW_HOW_PROTECT
//T10_T15,M0.2_M1.1,M10.0_M10.3,KA1_KA3
//
AUTHOR : NUMERIK
FAMILY : _800D
NAME : Enable
VERSION : 0.1
BEGIN
NETWORK
TITLE = Emergency stop                        
      A     "EMG_Active";
      S     DB10.DBX 56.1;
      R     DB10.DBX 56.2;
      A     "Reset_Key";
      S     DB10.DBX 56.2;
      R     DB10.DBX 56.1;
      A     DB10.DBX 56.4;
      =     "Key_0";
      A     DB10.DBX 56.5;
      =     "Key_1";
      A     DB10.DBX 56.6;
      =     "Key_2";
      A     DB10.DBX 56.7;
      =     "Key_3";
NETWORK
TITLE = 上电上升沿、松开急停上升沿
      AN    M 500.1;
      S     "ONE";
      R     "ZERO";
      AN    "EMG_Active";
      FP    M 500.2;
      =     "EMG_FP";
      A     "ONE";
      FP    M 500.6;
      =     "ONE_FP";
      A     "ONE";
      R     "INC_1000_LED";
      R     "INC_10000_LED";
      R     DB11.DBX 2.3;
      R     DB11.DBX 2.4;
      R     DB31.DBX 5.3;
      R     DB31.DBX 5.4;
      R     DB32.DBX 5.3;
      R     DB32.DBX 5.4;
      R     DB33.DBX 5.3;
      R     DB33.DBX 5.4;
      A     "EMG_Active";
      R     "FeedEnable_LED";
      S     "FeedDisable_LED";
NETWORK
TITLE = System power on and power off sequence control
//System power on and power off sequence control
//(T10～T15)
      A     "ONE";
      L     S5T#5S;
      SD    "KT0";
      A     "-QF17_驱动电源";
      A     DB10.DBX 108.7;
      AN    "KT4";
      =     "KA1_9_48";
      A     "KA1_9_48";
      A     "EP_Ready";
      A     DB10.DBX 108.5;
      AN    "KT3";
      L     S5T#1S;
      SD    "KT1";
      A     "KT1";
      =     "KA2_9_63";
      A     "KA2_9_63";
      A     "OFF1_Ready";
      AN    "EMG_Active";
      L     S5T#1S;
      SD    "KT2";
      A     "KT2";
      =     "KA3_9_64";
      A     "EMG_Active";
      L     S5T#2S;
      SD    "KT3";
      L     S5T#3S;
      SD    "KT4";
      A     "ONE";
      L     S5T#5M;
      SD    "KT5";
NETWORK
TITLE = Pulse enable and ContrEnable control
//M0.2_M1.5,T15
      A     "EMG_Active";
      A     "KT0";
      =     DB2.DBX 180.0;
      AN    "-QF17_驱动电源";
      =     DB2.DBX 181.7;
      AN    "OFF1_Ready";
      A     "KT5";
      =     DB2.DBX 183.0;
      AN    "EP_Ready";
      A     "KT5";
      =     DB2.DBX 182.7;
      AN    "KA1_9_48";
      A     "KT5";
      =     DB2.DBX 186.6;
      A     "FeedEnable_LED";
      A     "KA10_水冷机";
      A     "KA3_9_64";
      A     DB10.DBX 56.2;
      AN    DB2.DBX 182.2;
      AN    DB2.DBX 184.0;
      AN    DB2.DBX 184.1;
      AN    DB2.DBX 184.2;
      AN    DB2.DBX 184.3;
      AN    DB2.DBX 184.4;
      AN    DB2.DBX 184.5;
      AN    DB2.DBX 184.6;
      AN    "Time_Lock_Active";
      =     "Feed_Enable_X";
      A     "Refpoint_Key";
      =     DB21.DBX 1.0;
      CALL  "Axis_Control" (
           Enable                   := "Feed_Enable_X",
           Axis_Enc_Num             := DB120.DBB 0,
           Axis_Plus_LimitSwitch    := "-SQ1_X+",
           Axis_Minus_LimitSwitch   := "-SQ2_X-",
           Axis_Ref_Switch          := FALSE,
           Axis_PositContr          := DB31.DBX 61.5,
           Run_Mode                 := DB11.DBX 7.2,
           Axis_1st_Ref_Active      := DB31.DBX 60.4,
           Axis_2nd_Ref_Active      := DB31.DBX 60.5,
           Axis_Limitactive         := DB120.DBD 60,
           Axis_PulseEnable         := DB31.DBX 21.7,
           Axis_ContrEnable         := DB31.DBX 2.1,
           Axis_PosMeas1            := DB31.DBX 1.5,
           Axis_PosMeas2            := DB31.DBX 1.6,
           Axis_ORactive            := DB31.DBX 1.7,
           Axis_Refactive           := "X_Ref_OK",
           Axis_BreakActive         := "X_break_On",
           Axis_Plus_Limit          := DB31.DBX 12.1,
           Axis_Minus_Limit         := DB31.DBX 12.0,
           Axis_refpoint            := DB31.DBX 12.7);
      A     "Feed_Enable_X";
      =     "Feed_Enable_Z";
      CALL  "Axis_Control" (
           Enable                   := "Feed_Enable_Z",
           Axis_Enc_Num             := DB120.DBB 1,
           Axis_Plus_LimitSwitch    := "-SQ3_Z+",
           Axis_Minus_LimitSwitch   := "-SQ4_Z-",
           Axis_Ref_Switch          := FALSE,
           Axis_PositContr          := DB32.DBX 61.5,
           Run_Mode                 := DB11.DBX 7.2,
           Axis_1st_Ref_Active      := DB32.DBX 60.4,
           Axis_2nd_Ref_Active      := DB32.DBX 60.5,
           Axis_Limitactive         := DB120.DBD 60,
           Axis_PulseEnable         := DB32.DBX 21.7,
           Axis_ContrEnable         := DB32.DBX 2.1,
           Axis_PosMeas1            := DB32.DBX 1.5,
           Axis_PosMeas2            := DB32.DBX 1.6,
           Axis_ORactive            := DB32.DBX 1.7,
           Axis_Refactive           := "Z_Ref_OK",
           Axis_BreakActive         := "Z_break_On",
           Axis_Plus_Limit          := DB32.DBX 12.1,
           Axis_Minus_Limit         := DB32.DBX 12.0,
           Axis_refpoint            := DB32.DBX 12.7);
      A     "Feed_Enable_X";
      =     "Feed_Enable_C";
      CALL  "Axis_Control" (
           Enable                   := "Feed_Enable_C",
           Axis_Enc_Num             := DB120.DBB 2,
           Axis_Plus_LimitSwitch    := TRUE,
           Axis_Minus_LimitSwitch   := TRUE,
           Axis_Ref_Switch          := FALSE,
           Axis_PositContr          := DB33.DBX 61.5,
           Run_Mode                 := DB11.DBX 7.2,
           Axis_1st_Ref_Active      := DB33.DBX 60.4,
           Axis_2nd_Ref_Active      := DB33.DBX 60.5,
           Axis_Limitactive         := DB120.DBD 60,
           Axis_PulseEnable         := DB33.DBX 21.7,
           Axis_ContrEnable         := DB33.DBX 2.1,
           Axis_PosMeas1            := DB33.DBX 1.5,
           Axis_PosMeas2            := DB33.DBX 1.6,
           Axis_ORactive            := DB33.DBX 1.7,
           Axis_Refactive           := "C_Ref_OK",
           Axis_BreakActive         := "C_break_On",
           Axis_Plus_Limit          := DB33.DBX 12.1,
           Axis_Minus_Limit         := DB33.DBX 12.0,
           Axis_refpoint            := DB33.DBX 12.7);
      AN    "X_Ref_OK";
      ON    "Z_Ref_OK";
      =     DB2.DBX 186.4;
      A     "Feed_A";
      AN    "Feed_B";
      AN    "Feed_C";
      AN    "Feed_D";
      AN    "Feed_E";
      =     DB2.DBX 186.5;
      BE;
END_FUNCTION

FUNCTION "All motors_ control" : VOID	// FC 31
TITLE = 电机控制
//KNOW_HOW_PROTECT
//M5.0_M9.9,M11.0_M14.0,KA4_KA14
//
VERSION : 0.0
BEGIN
NETWORK
TITLE = 手轮干涉控制
//M5.0_M5.2
      A(;
      O     DB11.DBX 6.0;
      O     DB11.DBX 6.1;
      );
      AN    "Reset_Key";
      AN    "T13_LED_X轴快退";
      AN    "INC_1000_LED";
      AN    "INC_10000_LED";
      AN    "INC_VAR_LED";
      =     M 5.0;
      CALL  "Single Key control" (
           CH1_M_ON                 := FALSE,
           CH2_M_ON                 := FALSE,
           CH1_M_OFF                := FALSE,
           CH2_M_OFF                := FALSE,
           Key                      := "T1_DRF",
           Var1                     := M 5.1,
           Var2                     := M 5.2,
           Var3_up                  := FALSE,
           Protect                  := M 5.0,
           KeyEnableMode            := TRUE,
           KA                       := "T1_LED_DRF",
           LED                      := "T1_LED_DRF");
      A     "T1_LED_DRF";
      =     DB21.DBX 0.3;
NETWORK
TITLE = 砂轮修整控制
//M5.3_M5.5
      AN    "Reset_Key";
      A     DB11.DBX 6.0;
      =     M 5.3;
      CALL  "Single Key control" (
           CH1_M_ON                 := FALSE,
           CH2_M_ON                 := FALSE,
           CH1_M_OFF                := FALSE,
           CH2_M_OFF                := FALSE,
           Key                      := "T2_修整",
           Var1                     := M 5.4,
           Var2                     := M 5.5,
           Var3_up                  := FALSE,
           Protect                  := M 5.3,
           KeyEnableMode            := TRUE,
           KA                       := "T2_LED_修整",
           LED                      := "T2_LED_修整");
      A     "T2_LED_修整";
      =     DB10.DBX 123.2;
NETWORK
TITLE = 砂轮主轴润滑泵、砂轮主轴电机启动/停止控制(KA16,KA27)
//M6.1_M6.3,T20,T21,T22,KA16,KA27
      AN    "-QF14_砂轮电机";
      =     DB2.DBX 181.4;
      AN    "-QF16_AR润滑泵";
      =     DB2.DBX 181.6;
      A     "-ALARM_制动单元报警";
      =     DB2.DBX 182.0;
      AN    "-ALARM_主轴变频器报警";
      =     DB2.DBX 182.5;
      A     "-ALARM_主轴温度报警";
      =     DB2.DBX 183.1;
      AN    "-KP_润滑液位检测";
      =     DB2.DBX 183.2;
      A     "FeedEnable_LED";
      A     DB10.DBX 56.2;
      AN    DB2.DBX 181.6;
      AN    DB2.DBX 183.2;
      =     M 6.1;
      A     "ONE_FP";
      L     C#1;
      S     C 0;
      R     M 14.1;
      A(;
      O     "EMG_FP";
      O     M 14.0;
      );
      AN    "KT22";
      A     M 6.1;
      AN    M 14.1;
      =     M 14.0;
      L     S5T#30M;
      SD    "KT22";
      CD    C 0;
      A     C 0;
      A     "KT22";
      S     M 14.1;
      CALL  "Single Key control" (
           CH1_M_ON                 := DB21.DBX 195.5,
           CH2_M_ON                 := FALSE,
           CH1_M_OFF                := DB21.DBX 195.7,
           CH2_M_OFF                := FALSE,
           Key                      := "T4_砂轮",
           Var1                     := M 6.2,
           Var2                     := M 6.3,
           Var3_up                  := FALSE,
           Protect                  := M 6.1,
           KeyEnableMode            := TRUE,
           KA                       := M 14.2,
           LED                      := M 14.2);
      A     M 14.2;
      L     S5T#10M;
      SD    "KT10";
      A(;
      O     M 14.0;
      O     M 14.2;
      );
      =     "KA27_主轴润滑";
      =     "KA29_主轴气路";
      A(;
      O     M 14.1;
      O     "KT10";
      );
      AN    DB2.DBX 181.4;
      AN    DB2.DBX 182.0;
      AN    DB2.DBX 182.5;
      AN    DB2.DBX 183.1;
      AN    DB2.DBX 183.5;
      AN    DB2.DBX 184.6;
      =     "KA16_砂轮启停";
      A     "KA29_主轴气路";
      AN    "-KP_润滑气压检测";
      =     DB2.DBX 183.5;
      A     "KA27_主轴润滑";
      AN    "KT12";
      L     S5T#500MS;
      SD    "KT11";
      A     "KA27_主轴润滑";
      A     "KT11";
      L     S5T#500MS;
      SD    "KT12";
      A     "KT11";
      O     "KA16_砂轮启停";
      =     "T4_LED_砂轮";
      A     "KA16_砂轮启停";
      =     DB10.DBX 123.3;
NETWORK
TITLE = 滚轮电机启动/停止控制(KA17,KA18,KA19)
//M6.4_M6.6,T23,KA17,KA18,KA19
      AN    "-QF15_滚轮电机";
      =     DB2.DBX 181.5;
      AN    "-ALARM_滚轮驱动器报警";
      =     DB2.DBX 182.6;
      A     DB10.DBX 56.2;
      AN    DB2.DBX 181.5;
      AN    DB2.DBX 182.6;
      =     M 6.4;
      CALL  "Single Key control" (
           CH1_M_ON                 := DB21.DBX 201.7,
           CH2_M_ON                 := FALSE,
           CH1_M_OFF                := DB21.DBX 202.1,
           CH2_M_OFF                := FALSE,
           Key                      := "T5_滚轮",
           Var1                     := M 6.5,
           Var2                     := M 6.6,
           Var3_up                  := FALSE,
           Protect                  := M 6.4,
           KeyEnableMode            := TRUE,
           KA                       := "KA19_滚轮启停",
           LED                      := "T5_LED_滚轮");
      A     "KA19_滚轮启停";
      L     S5T#10S;
      SF    "KT13";
      A     "KT13";
      =     "KA17_滚轮使能";
      A     "KA19_滚轮启停";
      =     DB10.DBX 123.4;
      A     "Reset_Key";
      =     "KA18_报警复位";
NETWORK
TITLE = 电柜空调控制(KA11)
//M6.7_M7.1,KA11
      AN    "-QF8_电柜空调";
      =     DB2.DBX 181.0;
      A     "KA11_空调";
      AN    "-ALARM_空调报警";
      =     DB2.DBX 182.3;
      A     "-SB0_急停按钮";
      A     "-SB1_辅助急停1";
      A     "-SB2_辅助急停2";
      AN    DB2.DBX 181.0;
      =     M 6.7;
      CALL  "Single Key control" (
           CH1_M_ON                 := DB21.DBX 197.2,
           CH2_M_ON                 := FALSE,
           CH1_M_OFF                := DB21.DBX 197.3,
           CH2_M_OFF                := FALSE,
           Key                      := "T6_空调",
           Var1                     := M 7.0,
           Var2                     := M 7.1,
           Var3_up                  := "EMG_FP",
           Protect                  := M 6.7,
           KeyEnableMode            := TRUE,
           KA                       := "KA11_空调",
           LED                      := "T6_LED_空调");
NETWORK
TITLE = 冷却泵1控制(KA6)
//M7.2_M7.4,KA6
      AN    "-QF3_冷却泵1";
      =     DB2.DBX 180.3;
      AN    "-QF9_冷却装置";
      =     DB2.DBX 181.1;
      A     "-KP_冷却油液位检测";
      =     DB2.DBX 182.4;
      A     "-KP_漏油检测";
      =     DB2.DBX 184.7;
      A     DB10.DBX 56.2;
      AN    DB2.DBX 180.3;
      AN    DB2.DBX 181.1;
      AN    DB2.DBX 182.4;
      =     M 7.2;
      CALL  "Single Key control" (
           CH1_M_ON                 := DB21.DBX 195.0,
           CH2_M_ON                 := FALSE,
           CH1_M_OFF                := DB21.DBX 195.1,
           CH2_M_OFF                := FALSE,
           Key                      := "T7_冷却1",
           Var1                     := M 7.3,
           Var2                     := M 7.4,
           Var3_up                  := FALSE,
           Protect                  := M 7.2,
           KeyEnableMode            := TRUE,
           KA                       := "KA6_冷却泵1",
           LED                      := "T7_LED_冷却1");
NETWORK
TITLE = 冷却泵2控制(KA7)
//M7.5_M7.7,KA7
      AN    "-QF4_冷却泵2";
      =     DB2.DBX 180.4;
      A     DB10.DBX 56.2;
      AN    DB2.DBX 180.4;
      AN    DB2.DBX 181.1;
      AN    DB2.DBX 182.4;
      =     M 7.5;
      CALL  "Single Key control" (
           CH1_M_ON                 := DB21.DBX 197.4,
           CH2_M_ON                 := FALSE,
           CH1_M_OFF                := DB21.DBX 197.5,
           CH2_M_OFF                := FALSE,
           Key                      := "T8_冷却2",
           Var1                     := M 7.6,
           Var2                     := M 7.7,
           Var3_up                  := FALSE,
           Protect                  := M 7.5,
           KeyEnableMode            := TRUE,
           KA                       := "KA7_冷却泵2",
           LED                      := "T8_LED_冷却2");
NETWORK
TITLE = 冷却泵3控制(KA8)
//M8.0_M8.2,KA8
      AN    "-QF5_冷却泵3";
      =     DB2.DBX 180.5;
      A     DB10.DBX 56.2;
      AN    DB2.DBX 180.5;
      AN    DB2.DBX 181.1;
      AN    DB2.DBX 182.4;
      =     M 8.0;
      CALL  "Single Key control" (
           CH1_M_ON                 := DB21.DBX 198.6,
           CH2_M_ON                 := FALSE,
           CH1_M_OFF                := DB21.DBX 198.7,
           CH2_M_OFF                := FALSE,
           Key                      := "T9_冷却3",
           Var1                     := M 8.1,
           Var2                     := M 8.2,
           Var3_up                  := FALSE,
           Protect                  := M 8.0,
           KeyEnableMode            := TRUE,
           KA                       := "KA8_冷却泵3",
           LED                      := "T9_LED_冷却3");
NETWORK
TITLE = 液压头架夹紧/松开及液压泵控制(KA5,KA13,KA14,KA15)
//M8.3--M8.7,KA5,KA13,KA14,KA15
      AN    "-QF2_液压泵";
      =     DB2.DBX 180.2;
      A     "KA5_液压泵";
      AN    "-KP_液压油压力检测";
      =     DB2.DBX 183.3;
      AN    "EMG_Active";
      AN    DB2.DBX 180.2;
      =     M 8.3;
      CALL  "Single Key control" (
           CH1_M_ON                 := DB21.DBX 203.1,
           CH2_M_ON                 := FALSE,
           CH1_M_OFF                := DB21.DBX 203.2,
           CH2_M_OFF                := FALSE,
           Key                      := "T10_Һѹ",
           Var1                     := M 8.4,
           Var2                     := M 8.5,
           Var3_up                  := "EMG_FP",
           Protect                  := M 8.3,
           KeyEnableMode            := "JOG_LED",
           KA                       := "KA5_液压泵",
           LED                      := "T10_LED_Һѹ");
      AN    "KA5_液压泵";
      =     DB2.DBX 185.7;
      A(;
      A(;
      O     DB11.DBX 6.0;
      O     DB11.DBX 6.1;
      );
      A     DB21.DBX 35.7;
      O;
      A     DB11.DBX 6.2;
      AN    DB33.DBX 64.6;
      AN    DB33.DBX 64.7;
      );
      A     "-SF_脚踩开关";
      A     "KA5_液压泵";
      A     "KA23_门1打开";
      A     DB10.DBX 123.0;
      AN    DB2.DBX 183.3;
      =     M 8.6;
      A(;
      O     DB11.DBX 6.0;
      O     DB11.DBX 6.1;
      );
      A(;
      O     DB21.DBX 203.3;
      O     M 8.7;
      );
      AN    DB21.DBX 203.4;
      AN    DB33.DBX 64.7;
      AN    DB33.DBX 64.6;
      A     "KA5_液压泵";
      AN    DB2.DBX 183.3;
      =     M 8.7;
      A     M 8.6;
      O     M 8.7;
      =     "KA14_卡盘松开";
      AN    "KA14_卡盘松开";
      =     "KA13_卡盘夹紧";
      A     "KA13_卡盘夹紧";
      O     "KA14_卡盘松开";
      =     "KA15_卸荷阀";
      A     "-SQ6_卡盘夹紧到位";
      =     DB10.DBX 125.0;
      A     "-SQ5_卡盘松开到位";
      =     DB10.DBX 125.1;
NETWORK
TITLE = 吸雾器控制(KA9)
//M9.0_M9.2,KA9
      AN    "-QF6_吸雾器";
      =     DB2.DBX 180.6;
      A     DB10.DBX 56.2;
      AN    DB2.DBX 180.6;
      =     M 9.0;
      CALL  "Single Key control" (
           CH1_M_ON                 := DB21.DBX 196.4,
           CH2_M_ON                 := FALSE,
           CH1_M_OFF                := DB21.DBX 196.5,
           CH2_M_OFF                := FALSE,
           Key                      := "T11_吸雾",
           Var1                     := M 9.1,
           Var2                     := M 9.2,
           Var3_up                  := FALSE,
           Protect                  := M 9.0,
           KeyEnableMode            := TRUE,
           KA                       := "KA9_吸雾器",
           LED                      := "T11_LED_吸雾");
NETWORK
TITLE = 机床润滑控制(KA4)
//M9.3,T24,T25,T26,KA4
      AN    "-QF1_润滑泵";
      =     DB2.DBX 180.1;
      A     "-KP_润滑油液位检测";
      =     DB2.DBX 182.1;
      AN    "EMG_Active";
      AN    DB2.DBX 180.1;
      AN    DB2.DBX 182.1;
      =     M 9.3;
      A(;
      O     "T12_润滑";
      O     "EMG_FP";
      );
      A     M 9.3;
      L     S5T#10S;
      SF    "KT14";
      A     M 9.3;
      AN    "KT16";
      L     S5T#1H;
      SD    "KT15";
      A     M 9.3;
      A     "KT15";
      L     S5T#10S;
      SD    "KT16";
      A(;
      O     "KT14";
      O     "KT16";
      );
      A     M 9.3;
      =     "KA4_导轨润滑";
      =     "T12_LED_润滑";
NETWORK
TITLE = 机床照明灯控制(KA12)
//M9.4_M9.5,KA12
      CALL  "Single Key control" (
           CH1_M_ON                 := FALSE,
           CH2_M_ON                 := FALSE,
           CH1_M_OFF                := FALSE,
           CH2_M_OFF                := FALSE,
           Key                      := "T15_照明",
           Var1                     := M 9.4,
           Var2                     := M 9.5,
           Var3_up                  := "EMG_FP",
           Protect                  := TRUE,
           KeyEnableMode            := TRUE,
           KA                       := "KA12_照明灯",
           LED                      := "T15_LED_照明");
NETWORK
TITLE = C轴旋转控制
      A     DB11.DBX 6.0;
      A     "C_LED";
      =     DB10.DBX 1.5;
NETWORK
TITLE = 气动门1控制(KA23,KA24)
//M9.6_M9.7,M11.0_M11.3,M13.6,M13.7,KA23,KA24
//
      AN    "-KP_气压检测";
      =     DB2.DBX 183.4;
      CALL  "Single Key control" (
           CH1_M_ON                 := FALSE,
           CH2_M_ON                 := FALSE,
           CH1_M_OFF                := FALSE,
           CH2_M_OFF                := FALSE,
           Key                      := "9th_气动门锁强开",
           Var1                     := M 9.6,
           Var2                     := M 9.7,
           Var3_up                  := FALSE,
           Protect                  := DB21.DBX 35.0,
           KeyEnableMode            := DB11.DBX 6.0,
           KA                       := "9th_LED_强制打开",
           LED                      := "9th_LED_强制打开");
      A(;
      A(;
      O     DB11.DBX 6.0;
      O     DB11.DBX 6.1;
      );
      A     DB21.DBX 35.7;
      O     DB11.DBX 6.2;
      );
      A(;
      ON    "-KP_光幕1";
      O     "-KP_光幕2";
      );
      AN    DB10.DBX 123.0;
      =     M 13.6;
      A     DB10.DBX 56.2;
      AN    DB2.DBX 183.4;
      AN    M 13.6;
      AN    DB10.DBX 127.0;
      =     M 11.0;
      A(;
      A(;
      O     DB11.DBX 6.0;
      O     DB11.DBX 6.1;
      );
      A(;
      O     "9th_LED_强制打开";
      O     DB21.DBX 35.7;
      );
      O     DB11.DBX 6.2;
      );
      A     "7th_气动门1";
      AN    "KA16_砂轮启停";
      =     M 11.1;
      CALL  "Single Key control" (
           CH1_M_ON                 := DB21.DBX 200.0,
           CH2_M_ON                 := FALSE,
           CH1_M_OFF                := DB21.DBX 199.7,
           CH2_M_OFF                := FALSE,
           Key                      := M 11.1,
           Var1                     := M 11.2,
           Var2                     := M 11.3,
           Var3_up                  := FALSE,
           Protect                  := M 11.0,
           KeyEnableMode            := TRUE,
           KA                       := M 13.7,
           LED                      := M 13.7);
      AN    M 13.6;
      A     M 13.7;
      =     "KA24_门1关闭";
      A(;
      O     M 13.6;
      ON    M 13.7;
      );
      AN    "KA16_砂轮启停";
      AN    DB10.DBX 127.0;
      =     "KA23_门1打开";
      A     "ONE_FP";
      R     "7th_LED_气动门1";
      A     "-SQ7_左门1打开到位";
      A     "-SQ9_右门1打开到位";
      =     DB10.DBX 123.0;
      A     "-SQ8_左门1关闭到位";
      A     "-SQ10_右门1关闭到位";
      =     DB10.DBX 123.1;
      A     M 13.7;
      A     DB10.DBX 123.1;
      =     "7th_LED_气动门1";
NETWORK
TITLE = 气动门2控制(KA25,KA26)
//M11.4_M11.7,KA25,KA26
//
      A     DB10.DBX 56.2;
      AN    DB2.DBX 183.4;
      =     M 11.4;
      A(;
      A(;
      O     DB11.DBX 6.0;
      O     DB11.DBX 6.1;
      );
      A     "9th_LED_强制打开";
      O     DB11.DBX 6.2;
      );
      A     "8th_气动门2";
      =     M 11.5;
      CALL  "Single Key control" (
           CH1_M_ON                 := DB21.DBX 199.0,
           CH2_M_ON                 := FALSE,
           CH1_M_OFF                := DB21.DBX 198.5,
           CH2_M_OFF                := FALSE,
           Key                      := M 11.5,
           Var1                     := M 11.6,
           Var2                     := M 11.7,
           Var3_up                  := FALSE,
           Protect                  := M 11.4,
           KeyEnableMode            := TRUE,
           KA                       := "8th_LED_气动门2",
           LED                      := "8th_LED_气动门2");
      A     "8th_LED_气动门2";
      =     "KA26_门2关闭";
      AN    "8th_LED_气动门2";
      =     "KA25_门2打开";
      A     "ONE_FP";
      R     "8th_LED_气动门2";
      A     "-SQ11_左门2打开到位";
      A     "-SQ13_右门2打开到位";
      =     DB10.DBX 125.6;
      A     "-SQ12_左门2关闭到位";
      A     "-SQ14_右门2关闭到位";
      =     DB10.DBX 125.7;
NETWORK
TITLE = 机械锁控制(KA28)
//M12.0_M12.3,KA28
      A     DB10.DBX 56.2;
      =     M 12.0;
      A(;
      A(;
      O     DB11.DBX 6.0;
      O     DB11.DBX 6.1;
      );
      A     "9th_LED_强制打开";
      O     DB11.DBX 6.2;
      );
      A     "T14_机械门锁";
      =     M 12.1;
      CALL  "Single Key control" (
           CH1_M_ON                 := DB21.DBX 202.5,
           CH2_M_ON                 := FALSE,
           CH1_M_OFF                := DB21.DBX 202.2,
           CH2_M_OFF                := FALSE,
           Key                      := M 12.1,
           Var1                     := M 12.2,
           Var2                     := M 12.3,
           Var3_up                  := FALSE,
           Protect                  := M 12.0,
           KeyEnableMode            := TRUE,
           KA                       := "T14_LED_机械锁",
           LED                      := "T14_LED_机械锁");
      A     "T14_LED_机械锁";
      =     "KA28_机械门锁";
      A     "ONE_FP";
      R     "T14_LED_机械锁";
      A     "-LCCK_门锁状态1";
      A     "-LCCK_门锁状态2";
      AN    "-LCCK_门锁状态3";
      =     DB10.DBX 127.0;
NETWORK
TITLE = 手动对刀选择
//M12.4_M12.7,T16,T17
      A     DB11.DBX 6.0;
      AN    "T13_LED_X轴快退";
      AN    "Reset_Key";
      =     M 12.4;
      CALL  "Single Key control" (
           CH1_M_ON                 := FALSE,
           CH2_M_ON                 := FALSE,
           CH1_M_OFF                := FALSE,
           CH2_M_OFF                := FALSE,
           Key                      := "R10_手动对刀",
           Var1                     := M 12.5,
           Var2                     := M 12.6,
           Var3_up                  := FALSE,
           Protect                  := M 12.4,
           KeyEnableMode            := TRUE,
           KA                       := M 12.7,
           LED                      := M 12.7);
      A     M 12.7;
      =     DB10.DBX 1.0;
      A     M 12.7;
      AN    "KT7";
      L     S5T#500MS;
      SD    "KT6";
      A     M 12.7;
      A     "KT6";
      =     "R10_LED_手动对刀";
      A     M 12.7;
      A     "R10_LED_手动对刀";
      L     S5T#500MS;
      SD    "KT7";
NETWORK
TITLE = 自动对刀选择
//M13.0_M13.2,T18,T19
      CALL  "Single Key control" (
           CH1_M_ON                 := FALSE,
           CH2_M_ON                 := FALSE,
           CH1_M_OFF                := FALSE,
           CH2_M_OFF                := FALSE,
           Key                      := "R11_自动对刀",
           Var1                     := M 13.0,
           Var2                     := M 13.1,
           Var3_up                  := FALSE,
           Protect                  := M 12.4,
           KeyEnableMode            := TRUE,
           KA                       := M 13.2,
           LED                      := M 13.2);
      A     M 13.2;
      =     DB10.DBX 1.4;
      A     M 13.2;
      AN    "KT9";
      L     S5T#500MS;
      SD    "KT8";
      A     M 13.2;
      A     "KT8";
      =     "R11_LED_自动对刀";
      A     M 13.2;
      A     "R11_LED_自动对刀";
      L     S5T#500MS;
      SD    "KT9";
NETWORK
TITLE = 机床坐标系/工件坐标系转换
//M13.3_M13.5
      CALL  "Single Key control" (
           CH1_M_ON                 := FALSE,
           CH2_M_ON                 := FALSE,
           CH1_M_OFF                := FALSE,
           CH2_M_OFF                := FALSE,
           Key                      := "R12_工件坐标",
           Var1                     := M 13.3,
           Var2                     := M 13.4,
           Var3_up                  := FALSE,
           Protect                  := TRUE,
           KeyEnableMode            := TRUE,
           KA                       := M 13.5,
           LED                      := M 13.5);
      A     M 13.5;
      =     DB19.DBX 0.7;
      =     "R12_LED_工件坐标";
NETWORK
TITLE = 机械手控制
      CALL  "Truss manipulator" (
           IN0                      := "Input1_取成品到位",
           IN1                      := "Input2_送毛坯到位",
           IN2                      := "Input3_夹爪回到位",
           IN3                      := "Input4_备用1",
           IN4                      := "Input5_备用2",
           OUT0                     := "KA41_准备就绪",
           OUT1                     := "KA42_预完成",
           OUT2                     := "KA43_机械手故障",
           OUT3                     := "KA44_卡盘松开完成",
           OUT4                     := "KA45_卡盘夹紧完成",
           OUT5                     := "KA46_备用1",
           OUT6                     := "KA47_备用2",
           OUT7                     := "KA48_备用3");
NETWORK
TITLE = 机床水冷控制(KA10)
//KA10
      AN    "-QF7_水冷机";
      =     DB2.DBX 180.7;
      A     "KA10_水冷机";
      AN    "-ALARM_水冷机报警";
      =     DB2.DBX 182.2;
      A     "FeedEnable_LED";
      A     DB10.DBX 56.2;
      AN    DB2.DBX 180.7;
      =     "KA10_水冷机";
      AN    "-KP_水冷回路检测1";
      =     DB2.DBX 184.0;
      AN    "-KP_水冷回路检测2";
      =     DB2.DBX 184.1;
      AN    "-KP_水冷回路检测3";
      =     DB2.DBX 184.2;
      AN    "-KP_水冷回路检测4";
      =     DB2.DBX 184.3;
      AN    "-KP_水冷回路检测5";
      =     DB2.DBX 184.4;
      AN    "-KP_水冷回路检测6";
      =     DB2.DBX 184.5;
      AN    "-KP_电主轴水冷回路检测";
      =     DB2.DBX 184.6;
      AN    "-QF10_直流电源";
      =     DB2.DBX 181.2;
      AN    "-QF11_控制变压器";
      =     DB2.DBX 181.3;
      A     "-KP_灭火装置";
      =     DB2.DBX 185.0;
      A     "-UPS_电池报警";
      =     DB2.DBX 185.1;
NETWORK
TITLE = 警示灯控制(KA20、KA21、KA22)
      A     DB2.DBX 180.0;
      O     DB2.DBX 180.1;
      O     DB2.DBX 180.2;
      O     DB2.DBX 180.3;
      O     DB2.DBX 180.4;
      O     DB2.DBX 180.5;
      O     DB2.DBX 180.6;
      O     DB2.DBX 180.7;
      O     DB2.DBX 181.0;
      O     DB2.DBX 181.1;
      O     DB2.DBX 181.2;
      O     DB2.DBX 181.3;
      O     DB2.DBX 181.4;
      O     DB2.DBX 181.5;
      O     DB2.DBX 181.6;
      O     DB2.DBX 181.7;
      O     DB2.DBX 182.0;
      O     DB2.DBX 182.1;
      O     DB2.DBX 182.2;
      O     DB2.DBX 182.3;
      O     DB2.DBX 182.4;
      O     DB2.DBX 182.5;
      O     DB2.DBX 182.6;
      O     DB2.DBX 182.7;
      O     DB2.DBX 183.0;
      O     DB2.DBX 183.1;
      O     DB2.DBX 183.2;
      O     DB2.DBX 183.3;
      O     DB2.DBX 183.4;
      O     DB2.DBX 183.5;
      O     DB2.DBX 183.6;
      O     DB2.DBX 183.7;
      O     DB2.DBX 184.0;
      O     DB2.DBX 184.1;
      O     DB2.DBX 184.2;
      O     DB2.DBX 184.3;
      O     DB2.DBX 184.4;
      O     DB2.DBX 184.5;
      O     DB2.DBX 184.6;
      O     DB2.DBX 184.7;
      O     DB2.DBX 185.0;
      O     DB2.DBX 185.1;
      O     DB2.DBX 185.2;
      O     DB2.DBX 185.3;
      O     DB2.DBX 185.4;
      O     DB2.DBX 185.5;
      O     DB2.DBX 185.6;
      O     DB2.DBX 185.7;
      O     DB2.DBX 186.0;
      O     DB2.DBX 186.1;
      O     DB2.DBX 186.2;
      O     DB2.DBX 186.3;
      O     DB2.DBX 186.4;
      O     DB2.DBX 186.5;
      O     DB2.DBX 186.6;
      O     DB2.DBX 186.7;
      O     DB2.DBX 187.0;
      O     DB2.DBX 187.1;
      O     DB2.DBX 187.2;
      O     DB2.DBX 187.3;
      O     DB2.DBX 187.4;
      O     DB2.DBX 187.5;
      =     "KA20_红色";
      AN    DB21.DBX 35.0;
      AN    "KA20_红色";
      =     "KA21_黄色";
      A     DB21.DBX 35.0;
      AN    "KA21_黄色";
      =     "KA22_绿色";
      A     "Reset_Key";
      R     DB2.DBX 0.0;
      R     DB2.DBX 0.1;
      R     DB2.DBX 0.2;
      R     DB2.DBX 0.3;
      R     DB2.DBX 0.4;
      R     DB2.DBX 0.5;
      R     DB2.DBX 0.6;
      R     DB2.DBX 0.7;
      R     DB2.DBX 1.0;
      R     DB2.DBX 1.1;
      R     DB2.DBX 1.2;
      R     DB2.DBX 1.3;
      R     DB2.DBX 1.4;
      R     DB2.DBX 1.5;
      R     DB2.DBX 1.6;
      R     DB2.DBX 1.7;
      R     DB2.DBX 2.0;
      R     DB2.DBX 2.1;
      R     DB2.DBX 2.2;
      R     DB2.DBX 2.3;
      R     DB2.DBX 2.4;
      R     DB2.DBX 2.5;
      R     DB2.DBX 2.6;
      R     DB2.DBX 2.7;
      R     DB2.DBX 3.0;
      R     DB2.DBX 3.1;
      R     DB2.DBX 3.2;
      R     DB2.DBX 3.3;
      R     DB2.DBX 3.4;
      R     DB2.DBX 3.5;
      R     DB2.DBX 3.6;
      R     DB2.DBX 3.7;
      R     DB2.DBX 180.0;
      R     DB2.DBX 180.1;
      R     DB2.DBX 180.2;
      R     DB2.DBX 180.3;
      R     DB2.DBX 180.4;
      R     DB2.DBX 180.5;
      R     DB2.DBX 180.6;
      R     DB2.DBX 180.7;
      R     DB2.DBX 181.0;
      R     DB2.DBX 181.1;
      R     DB2.DBX 181.2;
      R     DB2.DBX 181.3;
      R     DB2.DBX 181.4;
      R     DB2.DBX 181.5;
      R     DB2.DBX 181.6;
      R     DB2.DBX 181.7;
      R     DB2.DBX 182.0;
      R     DB2.DBX 182.1;
      R     DB2.DBX 182.2;
      R     DB2.DBX 182.3;
      R     DB2.DBX 182.4;
      R     DB2.DBX 182.5;
      R     DB2.DBX 182.6;
      R     DB2.DBX 182.7;
      R     DB2.DBX 183.0;
      R     DB2.DBX 183.1;
      R     DB2.DBX 183.2;
      R     DB2.DBX 183.3;
      R     DB2.DBX 183.4;
      R     DB2.DBX 183.5;
      R     DB2.DBX 183.6;
      R     DB2.DBX 183.7;
      R     DB2.DBX 184.0;
      R     DB2.DBX 184.1;
      R     DB2.DBX 184.2;
      R     DB2.DBX 184.3;
      R     DB2.DBX 184.4;
      R     DB2.DBX 184.5;
      R     DB2.DBX 184.6;
      R     DB2.DBX 184.7;
      R     DB2.DBX 185.0;
      R     DB2.DBX 185.1;
      R     DB2.DBX 185.2;
      R     DB2.DBX 185.3;
      R     DB2.DBX 185.4;
      R     DB2.DBX 185.5;
      R     DB2.DBX 185.6;
      R     DB2.DBX 185.7;
      R     DB2.DBX 186.0;
      R     DB2.DBX 186.1;
      R     DB2.DBX 186.2;
      R     DB2.DBX 186.3;
      R     DB2.DBX 186.4;
      R     DB2.DBX 186.5;
      R     DB2.DBX 186.6;
      R     DB2.DBX 186.7;
      R     DB2.DBX 187.0;
      R     DB2.DBX 187.1;
      R     DB2.DBX 187.2;
      R     DB2.DBX 187.3;
      R     DB2.DBX 187.4;
      R     DB2.DBX 187.5;
      BE;
END_FUNCTION

FUNCTION "NC AND PLC CHANGE DATA" : VOID	// FC 32
TITLE = Read all axes enc_num and A21_A24 plus and minus limit
//KNOW_HOW_PROTECT
//M150.0_M150.5,MW300,MW302,DB100,DB120,DB150,DB151
//
VERSION : 0.1
BEGIN
NETWORK
TITLE =
      A     DB10.DBX 108.7;
      S     M 150.0;
      A     M 150.0;
      AN    M 150.2;
      S     M 150.2;
      A     M 150.1;
      A     M 150.2;
      R     M 150.2;
      CALL  "GET" , DB 150 (
           DIX 0.0                  := M 150.2,
           DIW 2                    := 8,
           DIW 4                    := W#16#1002,
           DIW 6                    := 10,
           DIW 8                    := 100,
           DID 10                   := P#DBX 0.0,
           DIW 20                   := W#16#1002,
           DIW 22                   := 10,
           DIW 24                   := 100,
           DID 26                   := P#DBX 10.0,
           DIW 36                   := W#16#1002,
           DIW 38                   := 10,
           DIW 40                   := 100,
           DID 42                   := P#DBX 20.0,
           DIW 52                   := W#16#1002,
           DIW 54                   := 10,
           DIW 56                   := 100,
           DID 58                   := P#DBX 30.0,
           DIW 68                   := W#16#1002,
           DIW 70                   := 10,
           DIW 72                   := 100,
           DID 74                   := P#DBX 40.0,
           DIW 84                   := W#16#1002,
           DIW 86                   := 10,
           DIW 88                   := 100,
           DID 90                   := P#DBX 50.0,
           DIW 100                  := W#16#1002,
           DIW 102                  := 10,
           DIW 104                  := 100,
           DID 106                  := P#DBX 60.0,
           DIW 116                  := W#16#1002,
           DIW 118                  := 10,
           DIW 120                  := 100,
           DID 122                  := P#DBX 70.0,
           DIX 132.0                := M 150.2,
           DIX 132.1                := M 150.1,
           DIW 134                  := MW 300,
           DIW 136                  := W#16#1002,
           DIW 138                  := 1,
           DIW 140                  := 120,
           DID 142                  := P#DBX 0.0,
           DIW 146                  := W#16#1002,
           DIW 148                  := 1,
           DIW 150                  := 120,
           DID 152                  := P#DBX 1.0,
           DIW 156                  := W#16#1002,
           DIW 158                  := 1,
           DIW 160                  := 120,
           DID 162                  := P#DBX 2.0,
           DIW 166                  := W#16#1002,
           DIW 168                  := 1,
           DIW 170                  := 120,
           DID 172                  := P#DBX 3.0,
           DIW 176                  := W#16#1002,
           DIW 178                  := 1,
           DIW 180                  := 120,
           DID 182                  := P#DBX 4.0,
           DIW 186                  := W#16#1002,
           DIW 188                  := 1,
           DIW 190                  := 120,
           DID 192                  := P#DBX 5.0,
           DIW 196                  := W#16#1002,
           DIW 198                  := 1,
           DIW 200                  := 120,
           DID 202                  := P#DBX 6.0,
           DIW 206                  := W#16#1002,
           DIW 208                  := 1,
           DIW 210                  := 120,
           DID 212                  := P#DBX 7.0);
      A     DB10.DBX 108.7;
      S     M 150.3;
      A     M 150.3;
      AN    M 150.5;
      S     M 150.5;
      A     M 150.4;
      A     M 150.5;
      R     M 150.5;
      CALL  "GET" , DB 151 (
           DIX 0.0                  := M 150.5,
           DIW 2                    := 8,
           DIW 4                    := W#16#1002,
           DIW 6                    := 10,
           DIW 8                    := 100,
           DID 10                   := P#DBX 80.0,
           DIW 20                   := W#16#1002,
           DIW 22                   := 10,
           DIW 24                   := 100,
           DID 26                   := P#DBX 90.0,
           DIW 36                   := W#16#1002,
           DIW 38                   := 10,
           DIW 40                   := 100,
           DID 42                   := P#DBX 100.0,
           DIW 52                   := W#16#1002,
           DIW 54                   := 10,
           DIW 56                   := 100,
           DID 58                   := P#DBX 110.0,
           DIW 68                   := W#16#1002,
           DIW 70                   := 10,
           DIW 72                   := 100,
           DID 74                   := P#DBX 120.0,
           DIW 84                   := W#16#1002,
           DIW 86                   := 10,
           DIW 88                   := 100,
           DID 90                   := P#DBX 130.0,
           DIW 100                  := W#16#1002,
           DIW 102                  := 10,
           DIW 104                  := 100,
           DID 106                  := P#DBX 140.0,
           DIW 116                  := W#16#1002,
           DIW 118                  := 10,
           DIW 120                  := 100,
           DID 122                  := P#DBX 150.0,
           DIX 132.0                := M 150.5,
           DIX 132.1                := M 150.4,
           DIW 134                  := MW 302,
           DIW 136                  := W#16#1006,
           DIW 138                  := 1,
           DIW 140                  := 120,
           DID 142                  := P#DBX 10.0,
           DIW 146                  := W#16#1006,
           DIW 148                  := 1,
           DIW 150                  := 120,
           DID 152                  := P#DBX 20.0,
           DIW 156                  := W#16#1006,
           DIW 158                  := 1,
           DIW 160                  := 120,
           DID 162                  := P#DBX 30.0,
           DIW 166                  := W#16#1006,
           DIW 168                  := 1,
           DIW 170                  := 120,
           DID 172                  := P#DBX 40.0,
           DIW 176                  := W#16#1006,
           DIW 178                  := 1,
           DIW 180                  := 120,
           DID 182                  := P#DBX 50.0,
           DIW 186                  := W#16#1006,
           DIW 188                  := 1,
           DIW 190                  := 120,
           DID 192                  := P#DBX 60.0,
           DIW 196                  := W#16#1006,
           DIW 198                  := 1,
           DIW 200                  := 120,
           DID 202                  := P#DBX 70.0,
           DIW 206                  := W#16#1006,
           DIW 208                  := 1,
           DIW 210                  := 120,
           DID 212                  := P#DBX 80.0);	//砂轮电机最高转速 / 滚轮电机最高转速 / 砂轮最大直径 / 砂轮最小直径 / 滚轮直径 / 各进给轴硬限位及参考点开关是否有效(0:有效;1:无效) / 运行时间设定是否生效(0:无效;1:有效)  / 运行时间设定 
      A     "Reset_Key";
      R     M 150.2;
      R     M 150.5;
      BE;
END_FUNCTION

FUNCTION "HandWheelUnit_Control" : VOID	// FC 33
//KNOW_HOW_PROTECT
//
NAME : FLX
VERSION : 0.1
BEGIN
NETWORK
TITLE = 手持单元有效
      A(;
      O     "KT1_X51.1_L1";
      O     "KT2_X51.2_L2";
      );
      A(;
      O     "JOG_LED";
      O     "T1_LED_DRF";
      );
      O;
      A     "KT3_X51.3_L4";
      A     "JOG_LED";
      =     "*HHU";
      =     "KT_OUT3_X53.3";
      =     DB2.DBX 186.0;
      A     "*HHU";
      A     "ONE";
      JCN   END1;
NETWORK
TITLE = 手持单元有效
      A     "*HHU";
      A     "KT1_X51.1_L1";
      =     "*X";
      S     "X_LED";
      R     "Z_LED";
      R     "C_LED";
      A     "*HHU";
      A     "KT2_X51.2_L2";
      =     "*Z";
      S     "Z_LED";
      R     "X_LED";
      R     "C_LED";
      A     "*HHU";
      A     "KT3_X51.3_L4";
      =     "*C";
      S     "C_LED";
      R     "X_LED";
      R     "Z_LED";
      A     "*HHU";
      A     "KT4_X52.1_R1";
      =     "*1";
      A     "*HHU";
      A     "KT5_X52.2_R2";
      =     "*10";
      A     "*HHU";
      A     "KT6_X52.3_R4";
      =     "*100";
NETWORK
TITLE = 手轮轴选增量有效
      A     "ONE";
      =     L 0.0;
      A     L 0.0;
      A(;
      O     "*1";
      O     "*10";
      O     "*100";
      );
      =     L 0.1;
      A     L 0.1;
      A(;
      O     "JOG_LED";
      O     "T1_LED_DRF";
      );
      A     "*X";
      =     DB31.DBX 4.0;
      A     L 0.1;
      A(;
      O     "JOG_LED";
      O     "T1_LED_DRF";
      );
      A     "*Z";
      =     DB32.DBX 4.0;
      A     L 0.1;
      A     "JOG_LED";
      A     "*C";
      =     DB33.DBX 4.0;
      A     L 0.0;
      A     "*1";
      =     DB31.DBX 5.0;
      =     DB32.DBX 5.0;
      =     DB33.DBX 5.0;
      =     DB11.DBX 2.0;
      =     DB2.DBX 186.1;
      A     L 0.0;
      A     "*10";
      =     DB31.DBX 5.1;
      =     DB32.DBX 5.1;
      =     DB33.DBX 5.1;
      =     DB11.DBX 2.1;
      =     DB2.DBX 186.2;
      A     L 0.0;
      A     "*100";
      =     DB31.DBX 5.2;
      =     DB32.DBX 5.2;
      =     DB33.DBX 5.2;
      =     DB11.DBX 2.2;
      =     DB2.DBX 186.3;
NETWORK
TITLE = 手持无效
END1: AN    "*HHU";
      R     DB31.DBX 4.0;
      R     DB32.DBX 4.0;
      R     DB33.DBX 4.0;
      R     DB2.DBX 186.0;
      R     DB2.DBX 186.1;
      R     DB2.DBX 186.2;
      R     DB2.DBX 186.3;
      A     "*HHU";
      L     S5T#1S;
      SF    "KT18";
      AN    "KT18";
      JC    END0;
      A     "*HHU";
      FN    M 500.4;
      =     "HHU_FN";
      A     "HHU_FN";
      R     "X_LED";
      R     "Z_LED";
      R     "C_LED";
      A     "HHU_FN";
      A     "JOG_LED";
      =     DB11.DBX 0.2;
      A     "HHU_FN";
      A     "Auto_LED";
      =     DB11.DBX 0.0;
END0: BE;
END_FUNCTION

FUNCTION "Grinding_Speed_1" : VOID	// FC 34
TITLE = GrindingWheel and FinishingWheel speed to be calculated
//KNOW_HOW_PROTECT
//M152.0_M153.4,MW308_MW312,DB104,DB122,DB123,DB124,DB154,DB155,DB156
//
VERSION : 0.1
BEGIN
NETWORK
TITLE =
      A     DB10.DBX 108.7;
      S     M 152.0;
      A     M 152.0;
      AN    M 152.2;
      S     M 152.2;
      A     M 152.1;
      A     M 152.2;
      R     M 152.2;
      CALL  "GET" , DB 154 (
           DIX 0.0                  := M 152.2,
           DIW 2                    := 6,
           DIW 4                    := W#16#1002,
           DIW 6                    := 10,
           DIW 8                    := 104,
           DID 10                   := P#DBX 0.0,
           DIW 20                   := W#16#1002,
           DIW 22                   := 10,
           DIW 24                   := 104,
           DID 26                   := P#DBX 20.0,
           DIW 36                   := W#16#1002,
           DIW 38                   := 10,
           DIW 40                   := 104,
           DID 42                   := P#DBX 30.0,
           DIW 52                   := W#16#1002,
           DIW 54                   := 10,
           DIW 56                   := 104,
           DID 58                   := P#DBX 50.0,
           DIW 68                   := W#16#1002,
           DIW 70                   := 10,
           DIW 72                   := 104,
           DID 74                   := P#DBX 60.0,
           DIW 84                   := W#16#1002,
           DIW 86                   := 10,
           DIW 88                   := 104,
           DID 90                   := P#DBX 70.0,
           DIX 132.0                := M 152.2,
           DIX 132.1                := M 152.1,
           DIW 134                  := MW 308,
           DIW 136                  := W#16#1006,
           DIW 138                  := 1,
           DIW 140                  := 122,
           DID 142                  := P#DBX 0.0,
           DIW 146                  := W#16#1006,
           DIW 148                  := 1,
           DIW 150                  := 122,
           DID 152                  := P#DBX 10.0,
           DIW 156                  := W#16#1006,
           DIW 158                  := 1,
           DIW 160                  := 122,
           DID 162                  := P#DBX 20.0,
           DIW 166                  := W#16#1006,
           DIW 168                  := 1,
           DIW 170                  := 122,
           DID 172                  := P#DBX 30.0,
           DIW 176                  := W#16#1006,
           DIW 178                  := 1,
           DIW 180                  := 122,
           DID 182                  := P#DBX 40.0,
           DIW 186                  := W#16#1006,
           DIW 188                  := 1,
           DIW 190                  := 122,
           DID 192                  := P#DBX 50.0);	//砂轮当前直径 / 滚轮与滚轮电机速比 / 滚轮与砂轮线速比 / 砂轮至砂轮电机速比 / 磨削时砂轮线速度 / 修整时砂轮线速度
NETWORK
TITLE =
      A     DB10.DBX 108.7;
      S     M 152.3;
      A     M 152.3;
      AN    M 152.5;
      S     M 152.5;
      A     M 152.4;
      A     M 152.5;
      R     M 152.5;
      CALL  "GET" , DB 155 (
           DIX 0.0                  := M 152.5,
           DIW 2                    := 5,
           DIW 4                    := W#16#1002,
           DIW 6                    := 10,
           DIW 8                    := 104,
           DID 10                   := P#DBX 110.0,
           DIW 20                   := W#16#1002,
           DIW 22                   := 10,
           DIW 24                   := 104,
           DID 26                   := P#DBX 120.0,
           DIW 36                   := W#16#1002,
           DIW 38                   := 10,
           DIW 40                   := 104,
           DID 42                   := P#DBX 130.0,
           DIW 52                   := W#16#1002,
           DIW 54                   := 10,
           DIW 56                   := 104,
           DID 58                   := P#DBX 140.0,
           DIW 68                   := W#16#1002,
           DIW 70                   := 10,
           DIW 72                   := 104,
           DID 74                   := P#DBX 150.0,
           DIX 132.0                := M 152.5,
           DIX 132.1                := M 152.4,
           DIW 134                  := MW 310,
           DIW 136                  := W#16#1006,
           DIW 138                  := 1,
           DIW 140                  := 122,
           DID 142                  := P#DBX 60.0,
           DIW 146                  := W#16#1006,
           DIW 148                  := 1,
           DIW 150                  := 122,
           DID 152                  := P#DBX 70.0,
           DIW 156                  := W#16#1006,
           DIW 158                  := 1,
           DIW 160                  := 122,
           DID 162                  := P#DBX 80.0,
           DIW 166                  := W#16#1006,
           DIW 168                  := 1,
           DIW 170                  := 122,
           DID 172                  := P#DBX 90.0,
           DIW 176                  := W#16#1006,
           DIW 178                  := 1,
           DIW 180                  := 122,
           DID 182                  := P#DBX 100.0);	//砂轮电机最高转速 / 滚轮电机最高转速 / 砂轮最大直径 / 砂轮最小直径 / 滚轮直径
NETWORK
TITLE =
      L     DB122.DBD 0;	//砂轮当前直径
      L     DB122.DBD 80;	//砂轮最大直径
      -R;
      JP    SPE0;
      L     DB122.DBD 90;	//砂轮最小直径
      L     DB122.DBD 0;	//砂轮当前直径
      -R;
      JP    SPE1;
      L     DB122.DBD 0;
      T     DB123.DBD 0;	//砂轮实际直径
      JU    SPE2;
SPE0: L     DB122.DBD 80;
      T     DB123.DBD 0;
      JU    SPE2;
SPE1: L     DB122.DBD 90;
      T     DB123.DBD 0;
SPE2: L     DB123.DBD 0;
      L     3.141593e+00;
      *R;
      T     DB123.DBD 10;
      L     DB122.DBD 40;	//磨削时砂轮线速度
      L     6.000000e+04;
      *R;
      T     DB123.DBD 20;
      L     DB123.DBD 20;
      L     DB123.DBD 10;
      /R;
      T     DB123.DBD 30;	//磨削时砂轮转速
      L     DB123.DBD 30;
      L     DB122.DBD 30;	//砂轮与电机传动比
      /R;
      T     DB123.DBD 40;	//磨削时砂轮电机转速
      L     DB123.DBD 40;
      L     DB122.DBD 60;
      -R;
      JP    SPE3;
      L     DB123.DBD 40;
      T     DB123.DBD 50;	//磨削时砂轮电机实际转速
      JU    SPE4;
SPE3: L     DB122.DBD 60;	//砂轮电机最高转速
      T     DB123.DBD 50;
//SPE4: L     DB122.DBD   70              //滚轮电机最高转速
//      L     DB122.DBD   10              //滚轮与滚轮电机速比
//      *R    
//      T     DB123.DBD   60              //滚轮最高转速
//     L     DB122.DBD  100              //滚轮直径
//      L     3.141593e+000
//      *R    
//     T     DB123.DBD   70
//     L     DB123.DBD   60
//     L     DB123.DBD   70
//      *R    
//      T     DB123.DBD   80
//      L     DB123.DBD   80
//     L     6.000000e+004
//      /R    
//      T     DB123.DBD   90              //滚轮最高线速度
//      L     DB122.DBD   50              //修整时砂轮线速度
//     L     DB122.DBD   20              //滚轮与砂轮线速比
//      *R    
//     T     DB123.DBD  100
//     L     DB123.DBD   90
//     L     DB123.DBD  100
//      -R    
//      JP    SPE5
//     L     DB123.DBD   90
//      T     DB123.DBD  110
//     JU    SPE6
//SPE5: L     DB123.DBD  100
//      T     DB123.DBD  110
//SPE6: L     DB123.DBD  110              //滚轮实际线速度
//     L     6.000000e+004
//      *R    
//      T     DB123.DBD  120
//      L     DB123.DBD  120
//      L     3.141593e+000
//      /R    
//      T     DB123.DBD  130
//      L     DB123.DBD  130
//      L     DB122.DBD  100
//      /R    
//      T     DB123.DBD  140              //滚轮实际转速
//      L     DB123.DBD  140
//      L     DB122.DBD   10
//      /R    
//     T     DB123.DBD  150              //滚轮电机实际转速
//     L     DB123.DBD  110
//     L     DB122.DBD   20
//      /R    
//      T     DB123.DBD  160              //修整时砂轮线速度
//      L     DB123.DBD  160
//     L     6.000000e+004
//      *R    
//     T     DB123.DBD  170
//      L     DB123.DBD  170
//     L     DB123.DBD   10
//      /R    
//      T     DB123.DBD  180
//      L     DB123.DBD  180
//      L     DB122.DBD   30
//      /R    
//      T     DB123.DBD  190
//      L     DB122.DBD   60
//      L     DB123.DBD  190
//      -R    
//      JP    SPE7
//      L     DB122.DBD   60
//      T     DB123.DBD  196              //修整时砂轮电机实际转速
//     JU    SPE8
//SPE7: L     DB123.DBD  190
//      T     DB123.DBD  196
//SPE8: L     DB123.DBD  196
//      L     DB122.DBD   30
//      *R    
//     T     DB124.DBD    0
//     L     DB124.DBD    0
//     L     DB123.DBD   10
//      *R    
//     T     DB124.DBD   10
//     L     DB124.DBD   10
//     L     6.000000e+004
//      /R    
//     T     DB124.DBD   20              //修整时砂轮实际线速度
NETWORK
TITLE = 模拟电压计算输出
//   AN    "T4_LED_砂轮"
//    A     "ONE"
//    JC    NET0
SPE4: L     DB123.DBD 50;
      T     DB124.DBD 30;
//      JU    NET1
//      L     DB123.DBD  196
//      T     DB124.DBD   30
//砂轮模拟电压输出计算
      L     DB124.DBD 30;
      L     DB122.DBD 60;
      /R;
      T     DB124.DBD 40;
      L     DB124.DBD 40;
      L     1.020000e+02;
      *R;
      T     DB124.DBD 50;
      L     DB124.DBD 50;
      TRUNC;
      T     DB124.DBD 60;
//滚轮模拟电压输出计算
      L     DB123.DBD 150;
      L     DB122.DBD 70;
      /R;
      T     DB124.DBD 70;
      L     DB124.DBD 70;
      L     1.020000e+02;
      *R;
      T     DB124.DBD 80;
      L     DB124.DBD 80;
      TRUNC;
      T     DB124.DBD 90;
//模拟电压输出
      L     B#16#55;
      T     QB 56;
      L     B#16#1;
      T     QB 57;
      L     "USER_DB4".STAT0[31];
      L     102;
      >=I;
      =     M 152.6;
      L     0;
      L     "USER_DB4".STAT0[31];
      >=I;
      =     M 152.7;
      A     "ONE";
      A     M 152.6;
      JC    SPP1;
      A     "ONE";
      A     M 152.7;
      JC    SPP2;
      L     "USER_DB4".STAT0[31];
      T     "USER_DB4".STAT0[50];
      JU    SPP3;
SPP1: L     102;
      T     "USER_DB4".STAT0[50];
      JU    SPP3;
SPP2: L     0;
      T     "USER_DB4".STAT0[50];
SPP3: L     "USER_DB4".STAT0[50];
      T     QW 60;	//模拟电压1输出
      L     "USER_DB4".STAT0[46];
      L     102;
      >=I;
      =     M 153.0;
      L     0;
      L     "USER_DB4".STAT0[46];
      >=I;
      =     M 153.1;
      A     "ONE";
      A     M 153.0;
      JC    SPP4;
      A     "ONE";
      A     M 153.1;
      JC    SPP5;
      L     "USER_DB4".STAT0[46];
      T     "USER_DB4".STAT0[51];
      JU    SPP6;
SPP4: L     102;
      T     "USER_DB4".STAT0[51];
      JU    SPP6;
SPP5: L     0;
      T     "USER_DB4".STAT0[51];
SPP6: L     "USER_DB4".STAT0[51];
      T     QW 62;	//模拟电压2输出 
NETWORK
TITLE = 砂轮电机、滚轮电机转速输出
      L     DB123.DBD 150;
      T     DB122.DBD 110;	//修整时滚轮电机转速
      L     DB123.DBD 110;
      T     DB122.DBD 120;	//修整时滚轮线速度
      L     DB123.DBD 50;
      T     DB122.DBD 130;	//磨削时砂轮电机转速
      L     DB123.DBD 196;
      T     DB122.DBD 140;	//修整时砂轮电机转速
      L     DB124.DBD 30;
      T     DB122.DBD 150;	//砂轮电机实际转速
      A     DB10.DBX 108.7;
      S     M 153.2;
      A     M 153.2;
      AN    M 153.4;
      S     M 153.4;
      A     M 153.3;
      A     M 153.4;
      R     M 153.4;
      CALL  "PUT" , DB 156 (
           DIX 0.0                  := M 153.4,
           DIW 2                    := 5,
           DIW 4                    := W#16#1002,
           DIW 6                    := 10,
           DIW 8                    := 104,
           DID 10                   := P#DBX 10.0,
           DIW 20                   := W#16#1002,
           DIW 22                   := 10,
           DIW 24                   := 104,
           DID 26                   := P#DBX 40.0,
           DIW 36                   := W#16#1002,
           DIW 38                   := 10,
           DIW 40                   := 104,
           DID 42                   := P#DBX 80.0,
           DIW 52                   := W#16#1002,
           DIW 54                   := 10,
           DIW 56                   := 104,
           DID 58                   := P#DBX 90.0,
           DIW 68                   := W#16#1002,
           DIW 70                   := 10,
           DIW 72                   := 104,
           DID 74                   := P#DBX 100.0,
           DIX 132.0                := M 153.4,
           DIX 132.1                := M 153.3,
           DIW 134                  := MW 312,
           DIW 136                  := W#16#1006,
           DIW 138                  := 1,
           DIW 140                  := 122,
           DID 142                  := P#DBX 110.0,
           DIW 146                  := W#16#1006,
           DIW 148                  := 1,
           DIW 150                  := 122,
           DID 152                  := P#DBX 120.0,
           DIW 156                  := W#16#1006,
           DIW 158                  := 1,
           DIW 160                  := 122,
           DID 162                  := P#DBX 130.0,
           DIW 166                  := W#16#1006,
           DIW 168                  := 1,
           DIW 170                  := 122,
           DID 172                  := P#DBX 140.0,
           DIW 176                  := W#16#1006,
           DIW 178                  := 1,
           DIW 180                  := 122,
           DID 182                  := P#DBX 150.0);	//滚轮电机转速 / 滚轮线速度 / 磨削时砂轮电机转速 / 修整时砂轮电机转速 / 砂轮电机实际转速
      A     "Reset_Key";
      R     M 152.2;
      R     M 152.5;
      R     M 153.4;
      BE;
END_FUNCTION

FUNCTION "Select program" : VOID	// FC 35
TITLE = Program select
//KNOW_HOW_PROTECT
//M154.0_M154.5,MW318,MW320,DB157,DB158
//
VERSION : 0.1
BEGIN
NETWORK
TITLE = Program to be selected
//M154.0_M154.5,MW318,MW320,DB157,DB158
      A     "T2_修整";	// Unassigned key on MCP
      A     DB11.DBX 6.7;
      S     M 154.0;	// Active Req
      A     M 154.2;	// Done message
      R     M 154.0;	// End job
      A     "Reset_Key";	// Acknowledge error manually
      A     M 154.1;	// Error is present
      R     M 154.0;
      A     M 154.0;
      S     "T2_LED_修整";
      R     "T3_LED_";
      CALL  "PI_SERV" , DB 157 (
           DIX 0.0                  := M 154.0,
           DIW 2                    := W#16#1002,
           DIW 4                    := 18,
           DIW 6                    := 16,
           DID 8                    := P#DBX 0.0,
           DIW 12                   := 1,
           DIW 14                   := W#16#1002,
           DIW 16                   := 34,
           DIW 18                   := 103,
           DID 20                   := P#DBX 34.0,
           DIW 24                   := W#16#1002,
           DIW 26                   := 34,
           DIW 28                   := 103,
           DID 30                   := P#DBX 0.0,
           DIX 74.0                 := M 154.1,
           DIX 74.1                 := M 154.2,
           DIW 76                   := MW 318);
      A     "T3_";
      A     DB11.DBX 6.7;
      S     M 154.3;
      A     M 154.5;	// Unassigned key on MCP
      R     M 154.3;
      A     "Reset_Key";	// Active Req
      A     M 154.4;	// Done message
      R     M 154.3;	// End job
      A     M 154.3;	// Acknowledge error manually
      S     "T3_LED_";	// Error is present
      R     "T2_LED_修整";
      CALL  "PI_SERV" , DB 158 (
           DIX 0.0                  := M 154.3,
           DIW 2                    := W#16#1002,
           DIW 4                    := 18,
           DIW 6                    := 16,
           DID 8                    := P#DBX 0.0,
           DIW 12                   := 1,
           DIW 14                   := W#16#1002,
           DIW 16                   := 34,
           DIW 18                   := 103,
           DID 20                   := P#DBX 102.0,
           DIW 24                   := W#16#1002,
           DIW 26                   := 34,
           DIW 28                   := 103,
           DID 30                   := P#DBX 68.0,
           DIX 74.0                 := M 154.4,
           DIX 74.1                 := M 154.5,
           DIW 76                   := MW 320);
      BE;
END_FUNCTION

FUNCTION "HandWheel_Control" : VOID	// FC 36
//KNOW_HOW_PROTECT
//
NAME : FLX
VERSION : 0.1
BEGIN
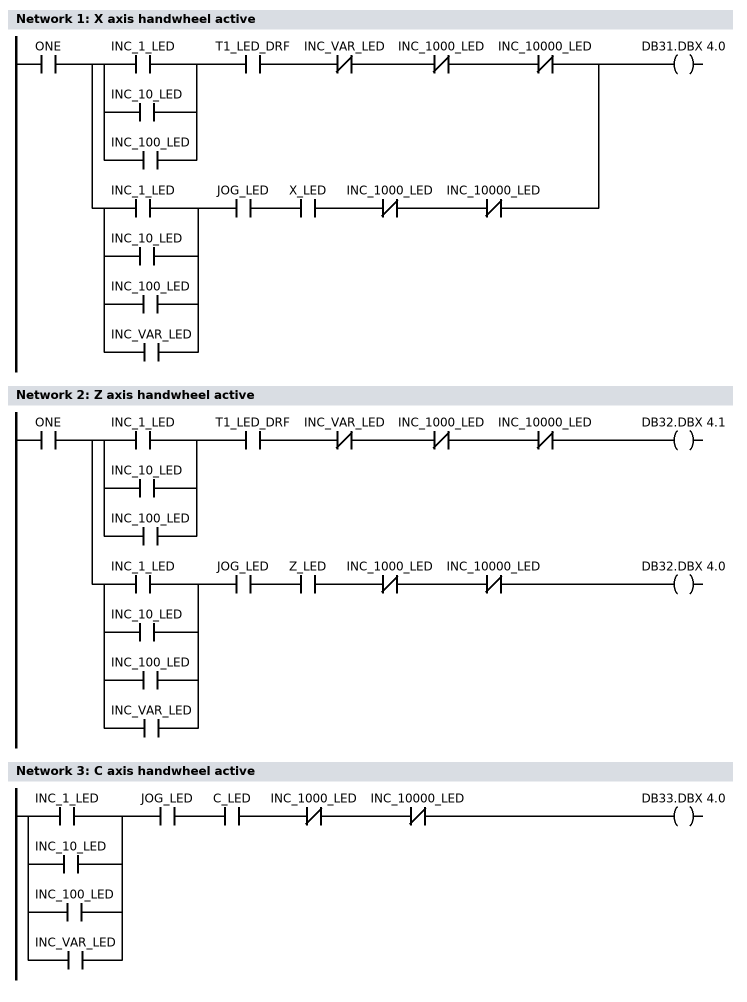
NETWORK
TITLE = X axis handwheel active
      A     "ONE";
      A(;
      A(;
      O     "INC_1_LED";
      O     "INC_10_LED";
      O     "INC_100_LED";
      );
      A     "T1_LED_DRF";
      AN    "INC_VAR_LED";
      AN    "INC_1000_LED";
      AN    "INC_10000_LED";
      O;
      A(;
      O     "INC_1_LED";
      O     "INC_10_LED";
      O     "INC_100_LED";
      O     "INC_VAR_LED";
      );
      A     "JOG_LED";
      A     "X_LED";
      AN    "INC_1000_LED";
      AN    "INC_10000_LED";
      );
      =     DB31.DBX 4.0;
NETWORK
TITLE = Z axis handwheel active
      A     "ONE";
      =     L 0.0;
      A     L 0.0;
      A(;
      O     "INC_1_LED";
      O     "INC_10_LED";
      O     "INC_100_LED";
      );
      A     "T1_LED_DRF";
      AN    "INC_VAR_LED";
      AN    "INC_1000_LED";
      AN    "INC_10000_LED";
      =     DB32.DBX 4.1;
      A     L 0.0;
      A(;
      O     "INC_1_LED";
      O     "INC_10_LED";
      O     "INC_100_LED";
      O     "INC_VAR_LED";
      );
      A     "JOG_LED";
      A     "Z_LED";
      AN    "INC_1000_LED";
      AN    "INC_10000_LED";
      =     DB32.DBX 4.0;
NETWORK
TITLE = C axis handwheel active
      A(;
      O     "INC_1_LED";
      O     "INC_10_LED";
      O     "INC_100_LED";
      O     "INC_VAR_LED";
      );
      A     "JOG_LED";
      A     "C_LED";
      AN    "INC_1000_LED";
      AN    "INC_10000_LED";
      =     DB33.DBX 4.0;
NETWORK
TITLE = 信息提示
      A     "T1_LED_DRF";
      =     DB2.DBX 186.0;
      A     "T1_LED_DRF";
      A     "INC_1_LED";
      =     DB2.DBX 186.1;
      A     "T1_LED_DRF";
      A     "INC_10_LED";
      =     DB2.DBX 186.2;
      A     "T1_LED_DRF";
      A     "INC_100_LED";
      =     DB2.DBX 186.3;
      BE;
END_FUNCTION

FUNCTION "Single Key control" : VOID	// FC 37
//KNOW_HOW_PROTECT
//
VERSION : 0.1
VAR_INPUT
  CH1_M_ON : BOOL ;	//The 1st chanel M code control motor running
  CH2_M_ON : BOOL ;	//The 2nd chanel M code control motor running
  CH1_M_OFF : BOOL ;	//The 1st chanel M code control motor stop
  CH2_M_OFF : BOOL ;	//The 2nd chanel M code control motor stop
  Key : BOOL ;	//Motor running orstopping control key
  Var1 : BOOL ;	//Var1
  Var2 : BOOL ;	//Var2
  Var3_up : BOOL ;	//Var3
  Protect : BOOL ;	//Motor protect
  KeyEnableMode : BOOL ;	//Mode_KeyEnable
END_VAR
VAR_OUTPUT
  KA : BOOL ;	//Output relay
  LED : BOOL ;	//Output led
END_VAR
BEGIN
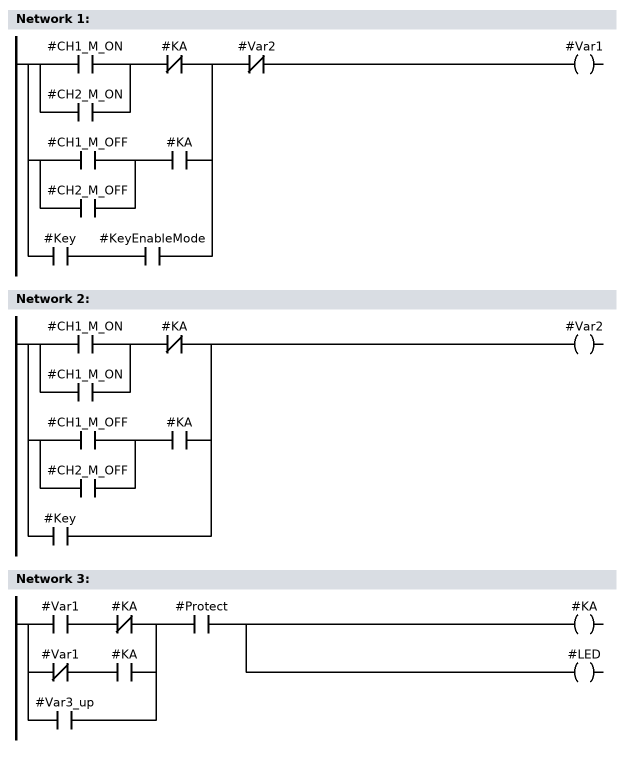
NETWORK
TITLE =
      A(;
      A(;
      O     #CH1_M_ON;
      O     #CH2_M_ON;
      );
      AN    #KA;
      O;
      A(;
      O     #CH1_M_OFF;
      O     #CH2_M_OFF;
      );
      A     #KA;
      O;
      A     #Key;
      A     #KeyEnableMode;
      );
      AN    #Var2;
      =     #Var1;
NETWORK
TITLE =
      A(;
      O     #CH1_M_ON;
      O     #CH1_M_ON;
      );
      AN    #KA;
      O;
      A(;
      O     #CH1_M_OFF;
      O     #CH2_M_OFF;
      );
      A     #KA;
      O     #Key;
      =     #Var2;
NETWORK
TITLE =
      A(;
      A     #Var1;
      AN    #KA;
      O;
      AN    #Var1;
      A     #KA;
      O     #Var3_up;
      );
      A     #Protect;
      =     #KA;
      =     #LED;
END_FUNCTION

